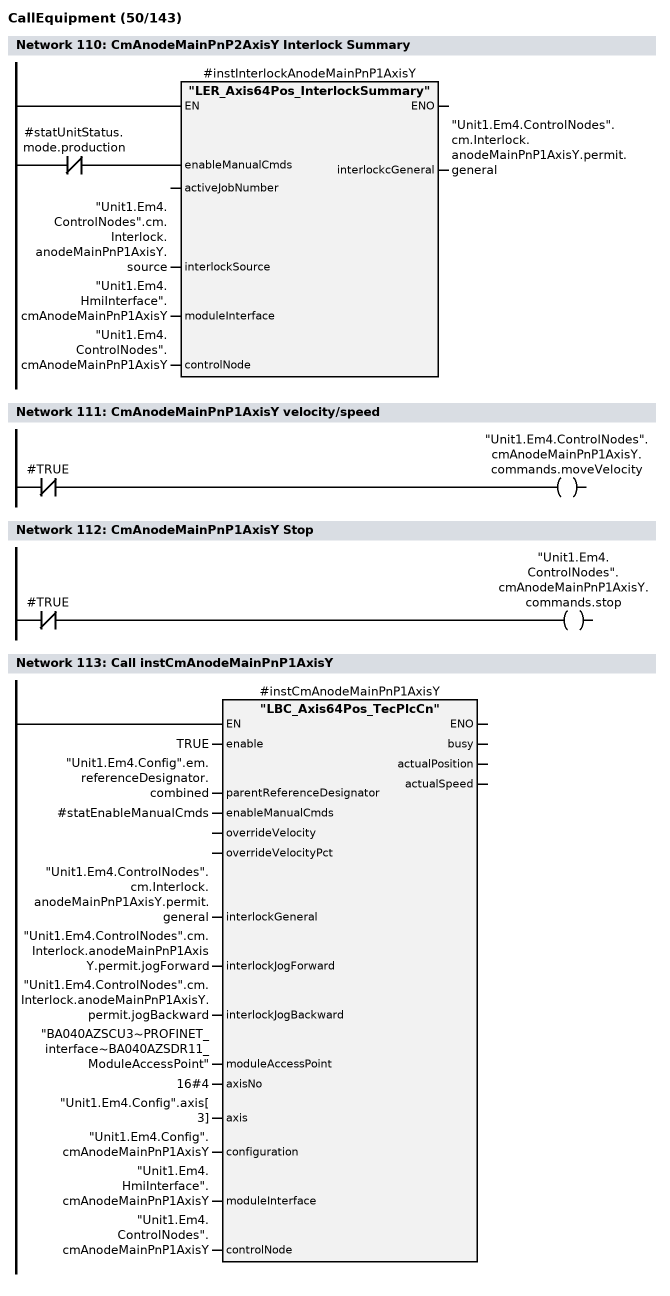
   RUNG wire#powerrail
      #instInterlockAnodeMainPnP1AxisY(enableManualCmds := wire#w1, activeJobNumber :=, interlockSource := "Unit1.Em4.ControlNodes".cm.Interlock.anodeMainPnP1AxisY.source, moduleInterface := "Unit1.Em4.HmiInterface".cmAnodeMainPnP1AxisY, controlNode := "Unit1.Em4.ControlNodes".cmAnodeMainPnP1AxisY, interlockcGeneral => "Unit1.Em4.ControlNodes".cm.Interlock.anodeMainPnP1AxisY.permit.general)
   END_RUNG
   RUNG wire#powerrail
      I_Contact( #statUnitStatus.mode.production )
   END_RUNG wire#w1
   // the same network as SCL:
   #instInterlockAnodeMainPnP1AxisY(enableManualCmds := NOT #statUnitStatus.mode.production,   // "LER_Axis64Pos_InterlockSummary"
                           interlockSource := "Unit1.Em4.ControlNodes".cm.Interlock.anodeMainPnP1AxisY.source,
                           moduleInterface := "Unit1.Em4.HmiInterface".cmAnodeMainPnP1AxisY,
                           controlNode := "Unit1.Em4.ControlNodes".cmAnodeMainPnP1AxisY,
                           interlockcGeneral => "Unit1.Em4.ControlNodes".cm.Interlock.anodeMainPnP1AxisY.permit.general);
END_REGION

REGION Network 111: CmAnodeMainPnP1AxisY velocity/speed
   RUNG wire#powerrail
      I_Contact( #TRUE )
      Coil( "Unit1.Em4.ControlNodes".cmAnodeMainPnP1AxisY.commands.moveVelocity )
   END_RUNG
   // the same network as SCL:
   "Unit1.Em4.ControlNodes".cmAnodeMainPnP1AxisY.commands.moveVelocity := NOT #TRUE;
END_REGION

REGION Network 112: CmAnodeMainPnP1AxisY Stop
   RUNG wire#powerrail
      I_Contact( #TRUE )
      Coil( "Unit1.Em4.ControlNodes".cmAnodeMainPnP1AxisY.commands.stop )
   END_RUNG
   // the same network as SCL:
   "Unit1.Em4.ControlNodes".cmAnodeMainPnP1AxisY.commands.stop := NOT #TRUE;
END_REGION

REGION Network 113: Call instCmAnodeMainPnP1AxisY
   RUNG wire#powerrail
      #instCmAnodeMainPnP1AxisY(enable := TRUE, parentReferenceDesignator := "Unit1.Em4.Config".em.referenceDesignator.combined, enableManualCmds := #statEnableManualCmds, overrideVelocity :=, overrideVelocityPct :=, interlockGeneral := "Unit1.Em4.ControlNodes".cm.Interlock.anodeMainPnP1AxisY.permit.general, interlockJogForward := "Unit1.Em4.ControlNodes".cm.Interlock.anodeMainPnP1AxisY.permit.jogForward, interlockJogBackward := "Unit1.Em4.ControlNodes".cm.Interlock.anodeMainPnP1AxisY.permit.jogBackward, moduleAccessPoint := "BA040AZSCU3~PROFINET_interface~BA040AZSDR11_ModuleAccessPoint", axisNo := 16#4, axis := "Unit1.Em4.Config".axis[3], configuration := "Unit1.Em4.Config".cmAnodeMainPnP1AxisY, moduleInterface := "Unit1.Em4.HmiInterface".cmAnodeMainPnP1AxisY, controlNode := "Unit1.Em4.ControlNodes".cmAnodeMainPnP1AxisY, busy =>, actualPosition =>, actualSpeed =>)
   END_RUNG
   // the same network as SCL:
   #instCmAnodeMainPnP1AxisY(enable := TRUE,   // "LBC_Axis64Pos_TecPlcCn"
                           parentReferenceDesignator := "Unit1.Em4.Config".em.referenceDesignator.combined,
                           enableManualCmds := #statEnableManualCmds,
                           interlockGeneral := "Unit1.Em4.ControlNodes".cm.Interlock.anodeMainPnP1AxisY.permit.general,
                           interlockJogForward := "Unit1.Em4.ControlNodes".cm.Interlock.anodeMainPnP1AxisY.permit.jogForward,
                           interlockJogBackward := "Unit1.Em4.ControlNodes".cm.Interlock.anodeMainPnP1AxisY.permit.jogBackward,
                           moduleAccessPoint := "BA040AZSCU3~PROFINET_interface~BA040AZSDR11_ModuleAccessPoint",
                           axisNo := 16#4,
                           axis := "Unit1.Em4.Config".axis[3],
                           configuration := "Unit1.Em4.Config".cmAnodeMainPnP1AxisY,
                           moduleInterface := "Unit1.Em4.HmiInterface".cmAnodeMainPnP1AxisY,
                           controlNode := "Unit1.Em4.ControlNodes".cmAnodeMainPnP1AxisY);
END_REGION

REGION Network 114: CmAnodeMainPnP1AxisY SoftCam
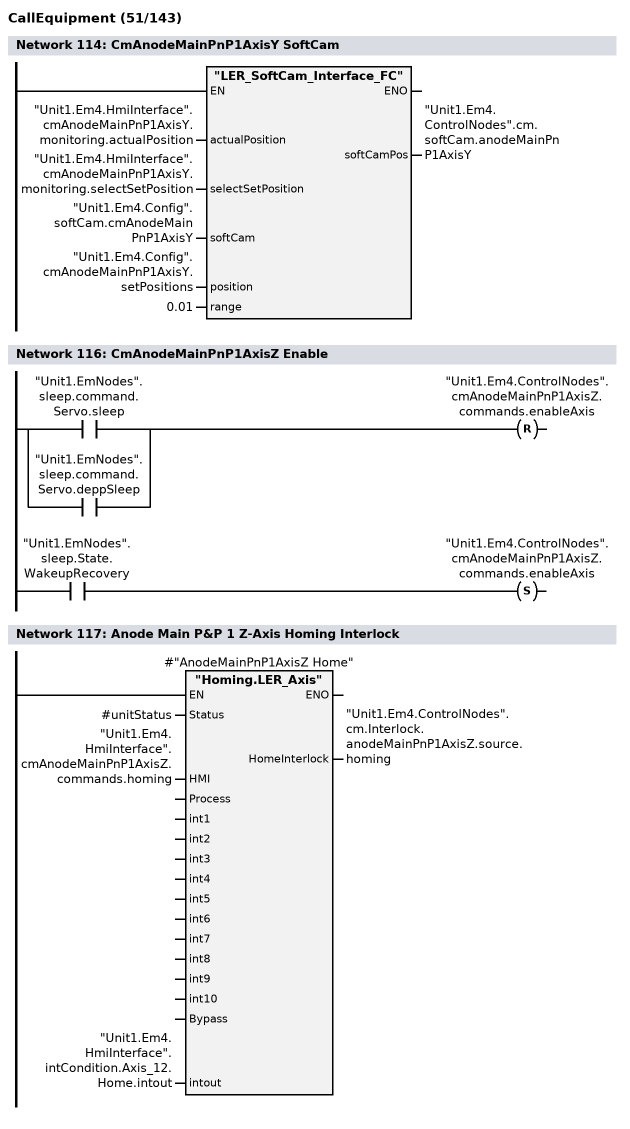
   RUNG wire#powerrail
      "LER_SoftCam_Interface_FC"(actualPosition := "Unit1.Em4.HmiInterface".cmAnodeMainPnP1AxisY.monitoring.actualPosition, selectSetPosition := "Unit1.Em4.HmiInterface".cmAnodeMainPnP1AxisY.monitoring.selectSetPosition, softCam := "Unit1.Em4.Config".softCam.cmAnodeMainPnP1AxisY, position := "Unit1.Em4.Config".cmAnodeMainPnP1AxisY.setPositions, range := 0.01, softCamPos => "Unit1.Em4.ControlNodes".cm.softCam.anodeMainPnP1AxisY)
   END_RUNG
   // the same network as SCL:
   "LER_SoftCam_Interface_FC"(actualPosition := "Unit1.Em4.HmiInterface".cmAnodeMainPnP1AxisY.monitoring.actualPosition,
                           selectSetPosition := "Unit1.Em4.HmiInterface".cmAnodeMainPnP1AxisY.monitoring.selectSetPosition,
                           softCam := "Unit1.Em4.Config".softCam.cmAnodeMainPnP1AxisY,
                           position := "Unit1.Em4.Config".cmAnodeMainPnP1AxisY.setPositions,
                           range := 0.01,
                           softCamPos => "Unit1.Em4.ControlNodes".cm.softCam.anodeMainPnP1AxisY);
END_REGION

REGION Network 116: CmAnodeMainPnP1AxisZ Enable
   RUNG wire#powerrail
      Contact( "Unit1.EmNodes".sleep.command.Servo.sleep )
      wire#w1
      R_Coil( "Unit1.Em4.ControlNodes".cmAnodeMainPnP1AxisZ.commands.enableAxis )
   END_RUNG
   RUNG wire#powerrail
      Contact( "Unit1.EmNodes".sleep.command.Servo.deppSleep )
   END_RUNG wire#w1
   RUNG wire#powerrail
      Contact( "Unit1.EmNodes".sleep.State.WakeupRecovery )
      S_Coil( "Unit1.Em4.ControlNodes".cmAnodeMainPnP1AxisZ.commands.enableAxis )
   END_RUNG
   // the same network as SCL:
   IF "Unit1.EmNodes".sleep.command.Servo.sleep OR "Unit1.EmNodes".sleep.command.Servo.deppSleep THEN
       "Unit1.Em4.ControlNodes".cmAnodeMainPnP1AxisZ.commands.enableAxis := FALSE;
   END_IF;
   IF "Unit1.EmNodes".sleep.State.WakeupRecovery THEN
       "Unit1.Em4.ControlNodes".cmAnodeMainPnP1AxisZ.commands.enableAxis := TRUE;
   END_IF;
END_REGION

REGION Network 117: Anode Main P&P 1 Z-Axis Homing Interlock
   RUNG wire#powerrail
      #"AnodeMainPnP1AxisZ Home"(Status := #unitStatus, HMI := "Unit1.Em4.HmiInterface".cmAnodeMainPnP1AxisZ.commands.homing, Process :=, int1 :=, int2 :=, int3 :=, int4 :=, int5 :=, int6 :=, int7 :=, int8 :=, int9 :=, int10 :=, Bypass :=, intout := "Unit1.Em4.HmiInterface".intCondition.Axis_12.Home.intout, HomeInterlock => "Unit1.Em4.ControlNodes".cm.Interlock.anodeMainPnP1AxisZ.source.homing)
   END_RUNG
   // the same network as SCL:
   #"AnodeMainPnP1AxisZ Home"(Status := #unitStatus,   // "Homing.LER_Axis"
                           HMI := "Unit1.Em4.HmiInterface".cmAnodeMainPnP1AxisZ.commands.homing,
                           intout := "Unit1.Em4.HmiInterface".intCondition.Axis_12.Home.intout,
                           HomeInterlock => "Unit1.Em4.ControlNodes".cm.Interlock.anodeMainPnP1AxisZ.source.homing);
END_REGION

REGION Network 118: CmAnodeMainPnP1AxisZ Position Absolute Jog
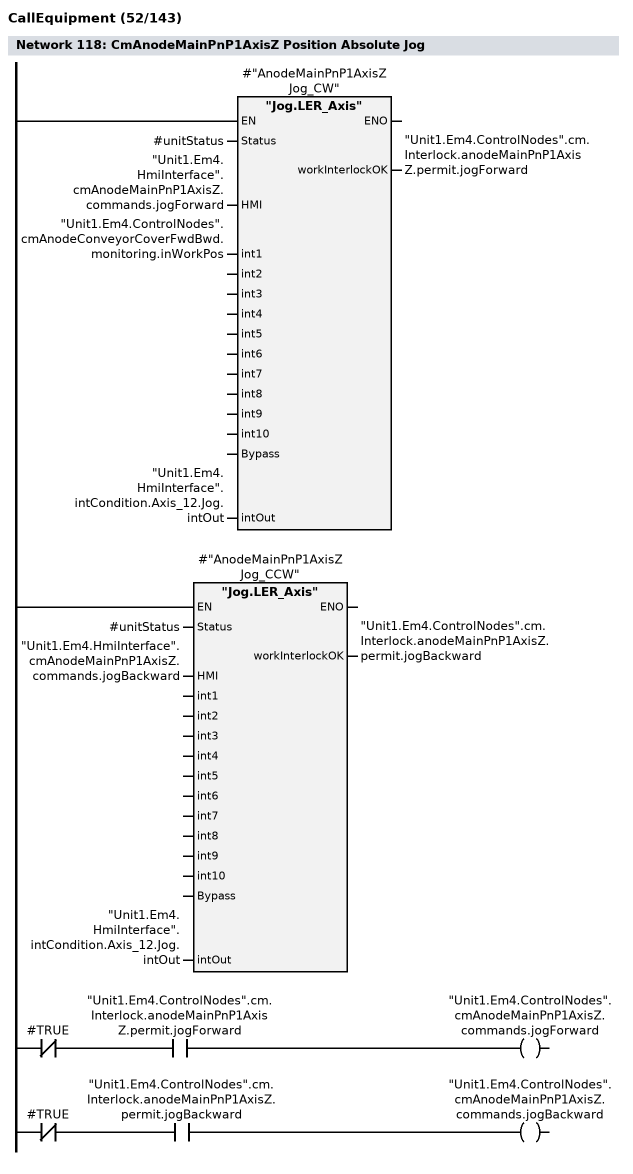
   RUNG wire#powerrail
      #"AnodeMainPnP1AxisZ Jog_CW"(Status := #unitStatus, HMI := "Unit1.Em4.HmiInterface".cmAnodeMainPnP1AxisZ.commands.jogForward, int1 := "Unit1.Em4.ControlNodes".cmAnodeConveyorCoverFwdBwd.monitoring.inWorkPos, int2 :=, int3 :=, int4 :=, int5 :=, int6 :=, int7 :=, int8 :=, int9 :=, int10 :=, Bypass :=, intOut := "Unit1.Em4.HmiInterface".intCondition.Axis_12.Jog.intOut, workInterlockOK => "Unit1.Em4.ControlNodes".cm.Interlock.anodeMainPnP1AxisZ.permit.jogForward)
   END_RUNG
   RUNG wire#powerrail
      #"AnodeMainPnP1AxisZ Jog_CCW"(Status := #unitStatus, HMI := "Unit1.Em4.HmiInterface".cmAnodeMainPnP1AxisZ.commands.jogBackward, int1 :=, int2 :=, int3 :=, int4 :=, int5 :=, int6 :=, int7 :=, int8 :=, int9 :=, int10 :=, Bypass :=, intOut := "Unit1.Em4.HmiInterface".intCondition.Axis_12.Jog.intOut, workInterlockOK => "Unit1.Em4.ControlNodes".cm.Interlock.anodeMainPnP1AxisZ.permit.jogBackward)
   END_RUNG
   RUNG wire#powerrail
      I_Contact( #TRUE )
      Contact( "Unit1.Em4.ControlNodes".cm.Interlock.anodeMainPnP1AxisZ.permit.jogForward )
      Coil( "Unit1.Em4.ControlNodes".cmAnodeMainPnP1AxisZ.commands.jogForward )
   END_RUNG
   RUNG wire#powerrail
      I_Contact( #TRUE )
      Contact( "Unit1.Em4.ControlNodes".cm.Interlock.anodeMainPnP1AxisZ.permit.jogBackward )
      Coil( "Unit1.Em4.ControlNodes".cmAnodeMainPnP1AxisZ.commands.jogBackward )
   END_RUNG
   // the same network as SCL:
   #"AnodeMainPnP1AxisZ Jog_CW"(Status := #unitStatus,   // "Jog.LER_Axis"
                           HMI := "Unit1.Em4.HmiInterface".cmAnodeMainPnP1AxisZ.commands.jogForward,
                           int1 := "Unit1.Em4.ControlNodes".cmAnodeConveyorCoverFwdBwd.monitoring.inWorkPos,
                           intOut := "Unit1.Em4.HmiInterface".intCondition.Axis_12.Jog.intOut,
                           workInterlockOK => "Unit1.Em4.ControlNodes".cm.Interlock.anodeMainPnP1AxisZ.permit.jogForward);
   #"AnodeMainPnP1AxisZ Jog_CCW"(Status := #unitStatus,   // "Jog.LER_Axis"
                           HMI := "Unit1.Em4.HmiInterface".cmAnodeMainPnP1AxisZ.commands.jogBackward,
                           intOut := "Unit1.Em4.HmiInterface".intCondition.Axis_12.Jog.intOut,
                           workInterlockOK => "Unit1.Em4.ControlNodes".cm.Interlock.anodeMainPnP1AxisZ.permit.jogBackward);
   "Unit1.Em4.ControlNodes".cmAnodeMainPnP1AxisZ.commands.jogForward := NOT #TRUE AND "Unit1.Em4.ControlNodes".cm.Interlock.anodeMainPnP1AxisZ.permit.jogForward;
   "Unit1.Em4.ControlNodes".cmAnodeMainPnP1AxisZ.commands.jogBackward := NOT #TRUE AND "Unit1.Em4.ControlNodes".cm.Interlock.anodeMainPnP1AxisZ.permit.jogBackward;
END_REGION

REGION Network 119: CmAnodeMainPnP1AxisZ Position Absolute Position0
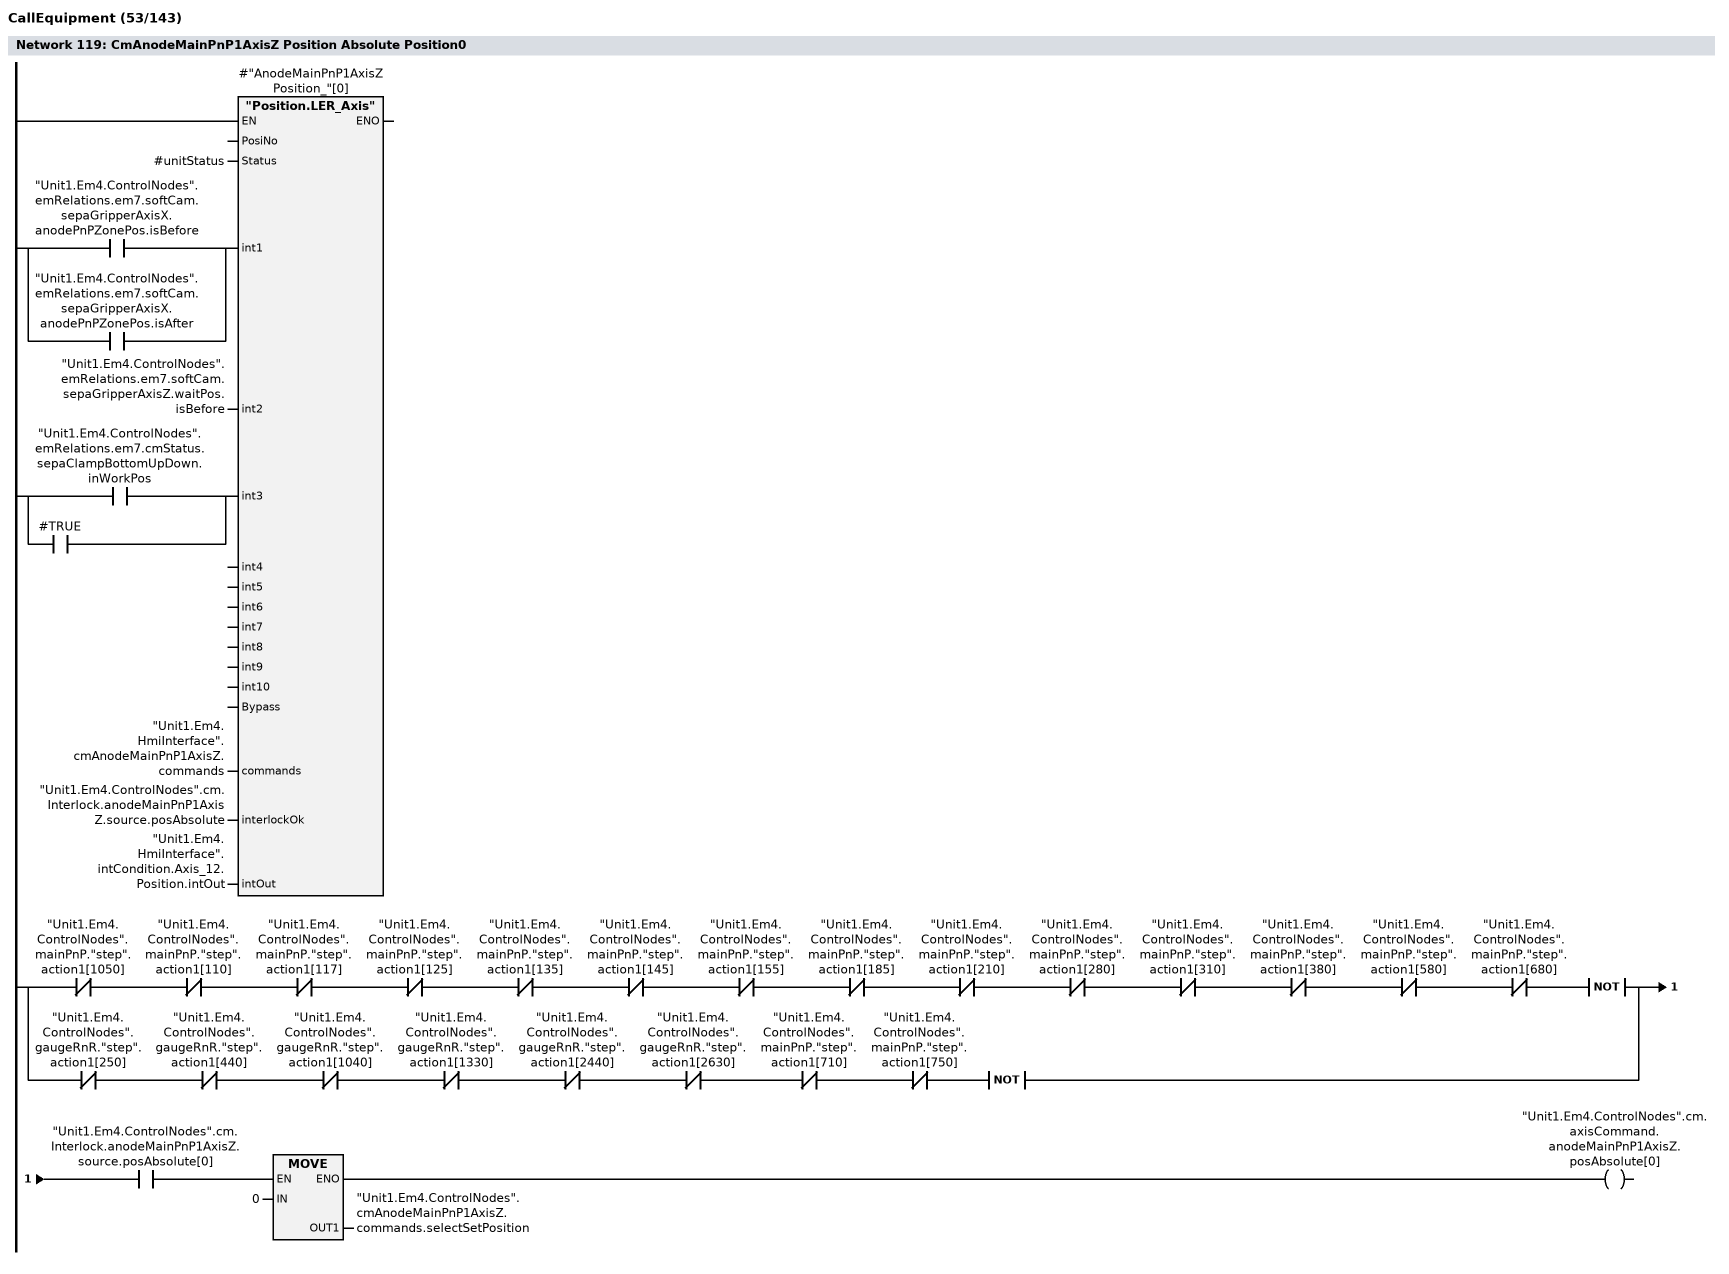
   RUNG wire#powerrail
      #"AnodeMainPnP1AxisZ Position_"[0](int1 := wire#w1, int3 := wire#w2, PosiNo :=, Status := #unitStatus, int2 := "Unit1.Em4.ControlNodes".emRelations.em7.softCam.sepaGripperAxisZ.waitPos.isBefore, int4 :=, int5 :=, int6 :=, int7 :=, int8 :=, int9 :=, int10 :=, Bypass :=, commands := "Unit1.Em4.HmiInterface".cmAnodeMainPnP1AxisZ.commands, interlockOk := "Unit1.Em4.ControlNodes".cm.Interlock.anodeMainPnP1AxisZ.source.posAbsolute, intOut := "Unit1.Em4.HmiInterface".intCondition.Axis_12.Position.intOut)
   END_RUNG
   RUNG wire#powerrail
      Contact( "Unit1.Em4.ControlNodes".emRelations.em7.softCam.sepaGripperAxisX.anodePnPZonePos.isBefore )
   END_RUNG wire#w1
   RUNG wire#powerrail
      Contact( "Unit1.Em4.ControlNodes".emRelations.em7.softCam.sepaGripperAxisX.anodePnPZonePos.isAfter )
   END_RUNG wire#w1
   RUNG wire#powerrail
      Contact( "Unit1.Em4.ControlNodes".emRelations.em7.cmStatus.sepaClampBottomUpDown.inWorkPos )
   END_RUNG wire#w2
   RUNG wire#powerrail
      Contact( #TRUE )
   END_RUNG wire#w2
   RUNG wire#powerrail
      I_Contact( "Unit1.Em4.ControlNodes".mainPnP."step".action1[1050] )
      I_Contact( "Unit1.Em4.ControlNodes".mainPnP."step".action1[110] )
      I_Contact( "Unit1.Em4.ControlNodes".mainPnP."step".action1[117] )
      I_Contact( "Unit1.Em4.ControlNodes".mainPnP."step".action1[125] )
      I_Contact( "Unit1.Em4.ControlNodes".mainPnP."step".action1[135] )
      I_Contact( "Unit1.Em4.ControlNodes".mainPnP."step".action1[145] )
      I_Contact( "Unit1.Em4.ControlNodes".mainPnP."step".action1[155] )
      I_Contact( "Unit1.Em4.ControlNodes".mainPnP."step".action1[185] )
      I_Contact( "Unit1.Em4.ControlNodes".mainPnP."step".action1[210] )
      I_Contact( "Unit1.Em4.ControlNodes".mainPnP."step".action1[280] )
      I_Contact( "Unit1.Em4.ControlNodes".mainPnP."step".action1[310] )
      I_Contact( "Unit1.Em4.ControlNodes".mainPnP."step".action1[380] )
      I_Contact( "Unit1.Em4.ControlNodes".mainPnP."step".action1[580] )
      I_Contact( "Unit1.Em4.ControlNodes".mainPnP."step".action1[680] )
      Not()
      wire#w3
      Contact( "Unit1.Em4.ControlNodes".cm.Interlock.anodeMainPnP1AxisZ.source.posAbsolute[0] )
      Move(in := 0, out1 => "Unit1.Em4.ControlNodes".cmAnodeMainPnP1AxisZ.commands.selectSetPosition)
      Coil( "Unit1.Em4.ControlNodes".cm.axisCommand.anodeMainPnP1AxisZ.posAbsolute[0] )
   END_RUNG
   RUNG wire#powerrail
      I_Contact( "Unit1.Em4.ControlNodes".gaugeRnR."step".action1[250] )
      I_Contact( "Unit1.Em4.ControlNodes".gaugeRnR."step".action1[440] )
      I_Contact( "Unit1.Em4.ControlNodes".gaugeRnR."step".action1[1040] )
      I_Contact( "Unit1.Em4.ControlNodes".gaugeRnR."step".action1[1330] )
      I_Contact( "Unit1.Em4.ControlNodes".gaugeRnR."step".action1[2440] )
      I_Contact( "Unit1.Em4.ControlNodes".gaugeRnR."step".action1[2630] )
      I_Contact( "Unit1.Em4.ControlNodes".mainPnP."step".action1[710] )
      I_Contact( "Unit1.Em4.ControlNodes".mainPnP."step".action1[750] )
      Not()
   END_RUNG wire#w3
   // the same network as SCL:
   #"AnodeMainPnP1AxisZ Position_"[0](Status := #unitStatus,   // "Position.LER_Axis"
                           int1 := "Unit1.Em4.ControlNodes".emRelations.em7.softCam.sepaGripperAxisX.anodePnPZonePos.isBefore OR "Unit1.Em4.ControlNodes".emRelations.em7.softCam.sepaGripperAxisX.anodePnPZonePos.isAfter,
                           int2 := "Unit1.Em4.ControlNodes".emRelations.em7.softCam.sepaGripperAxisZ.waitPos.isBefore,
                           int3 := "Unit1.Em4.ControlNodes".emRelations.em7.cmStatus.sepaClampBottomUpDown.inWorkPos OR #TRUE,
                           commands := "Unit1.Em4.HmiInterface".cmAnodeMainPnP1AxisZ.commands,
                           interlockOk := "Unit1.Em4.ControlNodes".cm.Interlock.anodeMainPnP1AxisZ.source.posAbsolute,
                           intOut := "Unit1.Em4.HmiInterface".intCondition.Axis_12.Position.intOut);
   #_w1 := (NOT (NOT "Unit1.Em4.ControlNodes".mainPnP."step".action1[1050] AND NOT "Unit1.Em4.ControlNodes".mainPnP."step".action1[110] AND NOT "Unit1.Em4.ControlNodes".mainPnP."step".action1[117] AND NOT "Unit1.Em4.ControlNodes".mainPnP."step".action1[125] AND NOT "Unit1.Em4.ControlNodes".mainPnP."step".action1[135] AND NOT "Unit1.Em4.ControlNodes".mainPnP."step".action1[145] AND NOT "Unit1.Em4.ControlNodes".mainPnP."step".action1[155] AND NOT "Unit1.Em4.ControlNodes".mainPnP."step".action1[185] AND NOT "Unit1.Em4.ControlNodes".mainPnP."step".action1[210] AND NOT "Unit1.Em4.ControlNodes".mainPnP."step".action1[280] AND NOT "Unit1.Em4.ControlNodes".mainPnP."step".action1[310] AND NOT "Unit1.Em4.ControlNodes".mainPnP."step".action1[380] AND NOT "Unit1.Em4.ControlNodes".mainPnP."step".action1[580] AND NOT "Unit1.Em4.ControlNodes".mainPnP."step".action1[680]) OR NOT (NOT "Unit1.Em4.ControlNodes".gaugeRnR."step".action1[250] AND NOT "Unit1.Em4.ControlNodes".gaugeRnR."step".action1[440] AND NOT "Unit1.Em4.ControlNodes".gaugeRnR."step".action1[1040] AND NOT "Unit1.Em4.ControlNodes".gaugeRnR."step".action1[1330] AND NOT "Unit1.Em4.ControlNodes".gaugeRnR."step".action1[2440] AND NOT "Unit1.Em4.ControlNodes".gaugeRnR."step".action1[2630] AND NOT "Unit1.Em4.ControlNodes".mainPnP."step".action1[710] AND NOT "Unit1.Em4.ControlNodes".mainPnP."step".action1[750])) AND "Unit1.Em4.ControlNodes".cm.Interlock.anodeMainPnP1AxisZ.source.posAbsolute[0];
   IF #_w1 THEN "Unit1.Em4.ControlNodes".cmAnodeMainPnP1AxisZ.commands.selectSetPosition := 0; END_IF;
   "Unit1.Em4.ControlNodes".cm.axisCommand.anodeMainPnP1AxisZ.posAbsolute[0] := #_w1;
END_REGION

REGION Network 120: CmAnodeMainPnP1AxisZ Position Absolute Position1
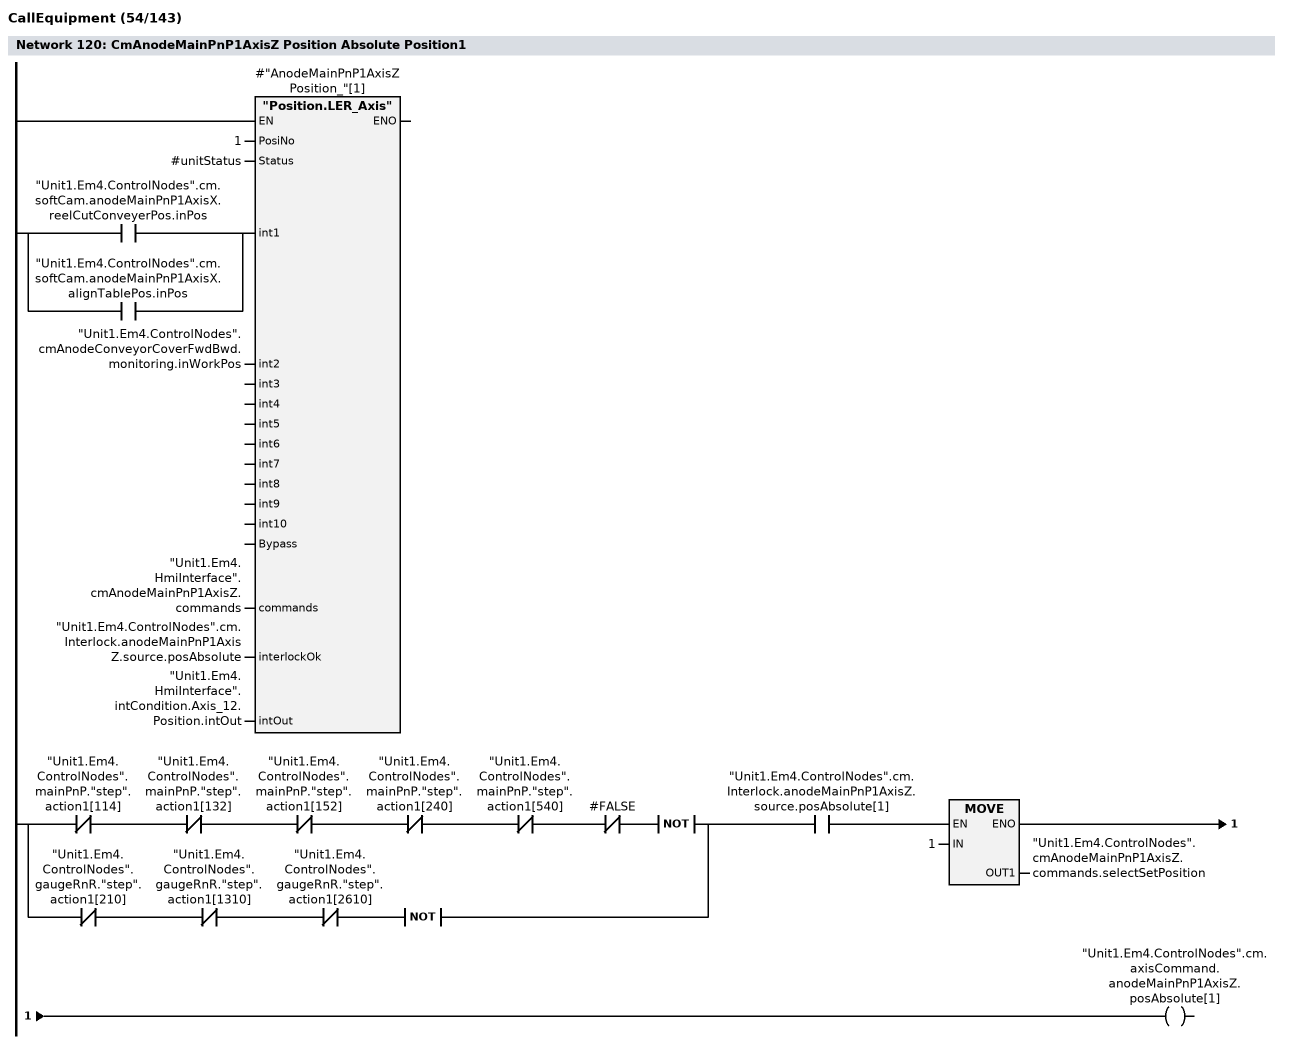
   RUNG wire#powerrail
      #"AnodeMainPnP1AxisZ Position_"[1](int1 := wire#w1, PosiNo := 1, Status := #unitStatus, int2 := "Unit1.Em4.ControlNodes".cmAnodeConveyorCoverFwdBwd.monitoring.inWorkPos, int3 :=, int4 :=, int5 :=, int6 :=, int7 :=, int8 :=, int9 :=, int10 :=, Bypass :=, commands := "Unit1.Em4.HmiInterface".cmAnodeMainPnP1AxisZ.commands, interlockOk := "Unit1.Em4.ControlNodes".cm.Interlock.anodeMainPnP1AxisZ.source.posAbsolute, intOut := "Unit1.Em4.HmiInterface".intCondition.Axis_12.Position.intOut)
   END_RUNG
   RUNG wire#powerrail
      Contact( "Unit1.Em4.ControlNodes".cm.softCam.anodeMainPnP1AxisX.reelCutConveyerPos.inPos )
   END_RUNG wire#w1
   RUNG wire#powerrail
      Contact( "Unit1.Em4.ControlNodes".cm.softCam.anodeMainPnP1AxisX.alignTablePos.inPos )
   END_RUNG wire#w1
   RUNG wire#powerrail
      I_Contact( "Unit1.Em4.ControlNodes".mainPnP."step".action1[114] )
      I_Contact( "Unit1.Em4.ControlNodes".mainPnP."step".action1[132] )
      I_Contact( "Unit1.Em4.ControlNodes".mainPnP."step".action1[152] )
      I_Contact( "Unit1.Em4.ControlNodes".mainPnP."step".action1[240] )
      I_Contact( "Unit1.Em4.ControlNodes".mainPnP."step".action1[540] )
      I_Contact( #FALSE )
      Not()
      wire#w2
      Contact( "Unit1.Em4.ControlNodes".cm.Interlock.anodeMainPnP1AxisZ.source.posAbsolute[1] )
      Move(in := 1, out1 => "Unit1.Em4.ControlNodes".cmAnodeMainPnP1AxisZ.commands.selectSetPosition)
      Coil( "Unit1.Em4.ControlNodes".cm.axisCommand.anodeMainPnP1AxisZ.posAbsolute[1] )
   END_RUNG
   RUNG wire#powerrail
      I_Contact( "Unit1.Em4.ControlNodes".gaugeRnR."step".action1[210] )
      I_Contact( "Unit1.Em4.ControlNodes".gaugeRnR."step".action1[1310] )
      I_Contact( "Unit1.Em4.ControlNodes".gaugeRnR."step".action1[2610] )
      Not()
   END_RUNG wire#w2
   // the same network as SCL:
   #"AnodeMainPnP1AxisZ Position_"[1](PosiNo := 1,   // "Position.LER_Axis"
                           Status := #unitStatus,
                           int1 := "Unit1.Em4.ControlNodes".cm.softCam.anodeMainPnP1AxisX.reelCutConveyerPos.inPos OR "Unit1.Em4.ControlNodes".cm.softCam.anodeMainPnP1AxisX.alignTablePos.inPos,
                           int2 := "Unit1.Em4.ControlNodes".cmAnodeConveyorCoverFwdBwd.monitoring.inWorkPos,
                           commands := "Unit1.Em4.HmiInterface".cmAnodeMainPnP1AxisZ.commands,
                           interlockOk := "Unit1.Em4.ControlNodes".cm.Interlock.anodeMainPnP1AxisZ.source.posAbsolute,
                           intOut := "Unit1.Em4.HmiInterface".intCondition.Axis_12.Position.intOut);
   #_w1 := (NOT (NOT "Unit1.Em4.ControlNodes".mainPnP."step".action1[114] AND NOT "Unit1.Em4.ControlNodes".mainPnP."step".action1[132] AND NOT "Unit1.Em4.ControlNodes".mainPnP."step".action1[152] AND NOT "Unit1.Em4.ControlNodes".mainPnP."step".action1[240] AND NOT "Unit1.Em4.ControlNodes".mainPnP."step".action1[540] AND NOT #FALSE) OR NOT (NOT "Unit1.Em4.ControlNodes".gaugeRnR."step".action1[210] AND NOT "Unit1.Em4.ControlNodes".gaugeRnR."step".action1[1310] AND NOT "Unit1.Em4.ControlNodes".gaugeRnR."step".action1[2610])) AND "Unit1.Em4.ControlNodes".cm.Interlock.anodeMainPnP1AxisZ.source.posAbsolute[1];
   IF #_w1 THEN "Unit1.Em4.ControlNodes".cmAnodeMainPnP1AxisZ.commands.selectSetPosition := 1; END_IF;
   "Unit1.Em4.ControlNodes".cm.axisCommand.anodeMainPnP1AxisZ.posAbsolute[1] := #_w1;
END_REGION

REGION Network 121: CmAnodeMainPnP1AxisZ Position Absolute Position2
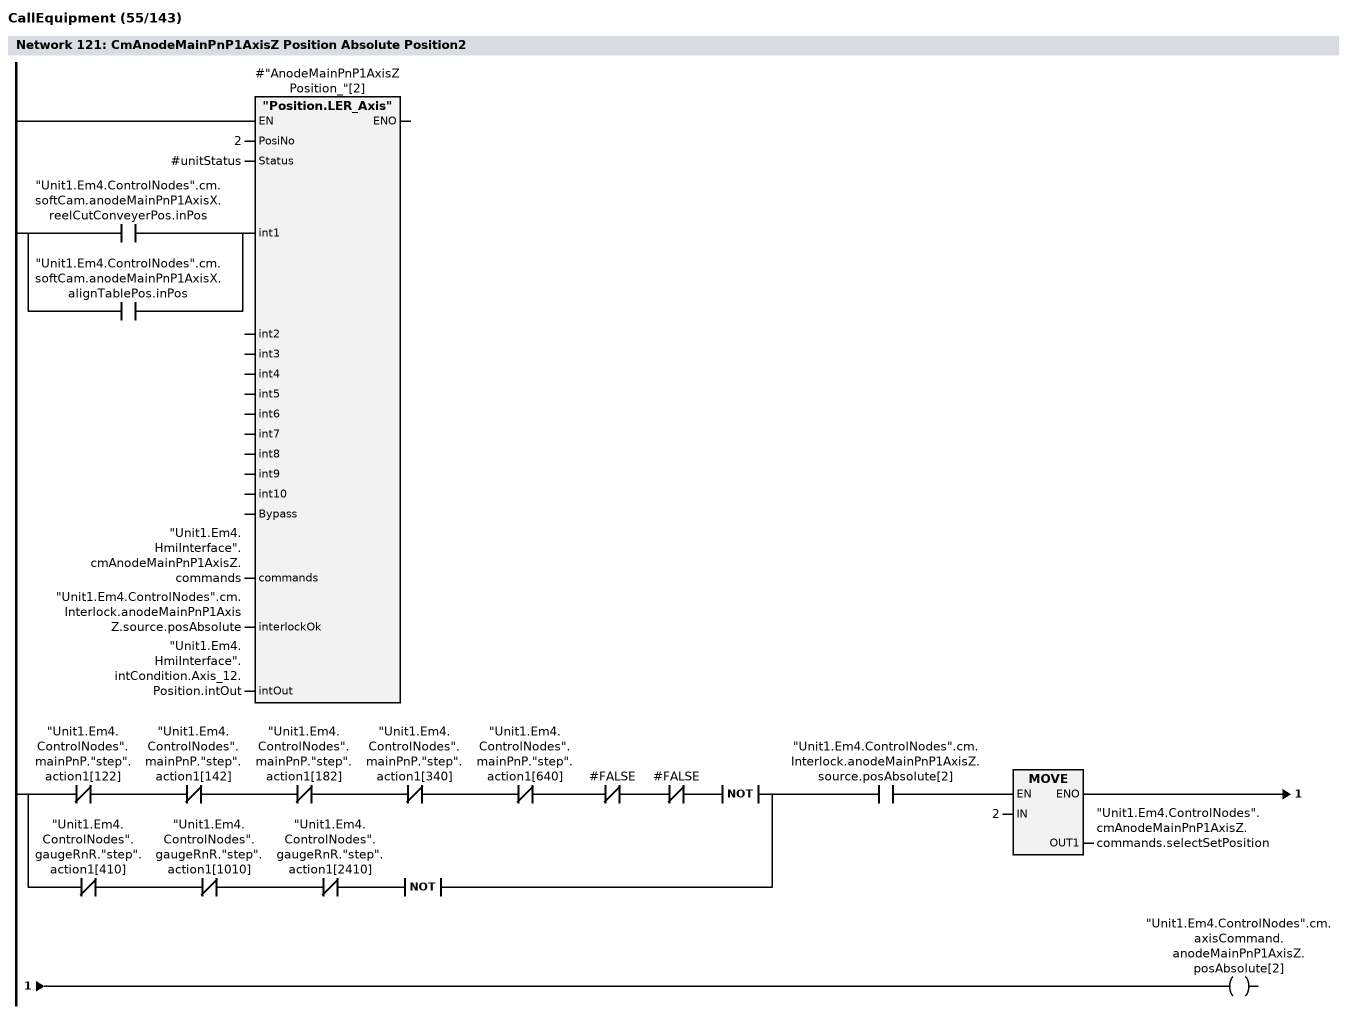
   RUNG wire#powerrail
      #"AnodeMainPnP1AxisZ Position_"[2](int1 := wire#w1, PosiNo := 2, Status := #unitStatus, int2 :=, int3 :=, int4 :=, int5 :=, int6 :=, int7 :=, int8 :=, int9 :=, int10 :=, Bypass :=, commands := "Unit1.Em4.HmiInterface".cmAnodeMainPnP1AxisZ.commands, interlockOk := "Unit1.Em4.ControlNodes".cm.Interlock.anodeMainPnP1AxisZ.source.posAbsolute, intOut := "Unit1.Em4.HmiInterface".intCondition.Axis_12.Position.intOut)
   END_RUNG
   RUNG wire#powerrail
      Contact( "Unit1.Em4.ControlNodes".cm.softCam.anodeMainPnP1AxisX.reelCutConveyerPos.inPos )
   END_RUNG wire#w1
   RUNG wire#powerrail
      Contact( "Unit1.Em4.ControlNodes".cm.softCam.anodeMainPnP1AxisX.alignTablePos.inPos )
   END_RUNG wire#w1
   RUNG wire#powerrail
      I_Contact( "Unit1.Em4.ControlNodes".mainPnP."step".action1[122] )
      I_Contact( "Unit1.Em4.ControlNodes".mainPnP."step".action1[142] )
      I_Contact( "Unit1.Em4.ControlNodes".mainPnP."step".action1[182] )
      I_Contact( "Unit1.Em4.ControlNodes".mainPnP."step".action1[340] )
      I_Contact( "Unit1.Em4.ControlNodes".mainPnP."step".action1[640] )
      I_Contact( #FALSE )
      I_Contact( #FALSE )
      Not()
      wire#w2
      Contact( "Unit1.Em4.ControlNodes".cm.Interlock.anodeMainPnP1AxisZ.source.posAbsolute[2] )
      Move(in := 2, out1 => "Unit1.Em4.ControlNodes".cmAnodeMainPnP1AxisZ.commands.selectSetPosition)
      Coil( "Unit1.Em4.ControlNodes".cm.axisCommand.anodeMainPnP1AxisZ.posAbsolute[2] )
   END_RUNG
   RUNG wire#powerrail
      I_Contact( "Unit1.Em4.ControlNodes".gaugeRnR."step".action1[410] )
      I_Contact( "Unit1.Em4.ControlNodes".gaugeRnR."step".action1[1010] )
      I_Contact( "Unit1.Em4.ControlNodes".gaugeRnR."step".action1[2410] )
      Not()
   END_RUNG wire#w2
   // the same network as SCL:
   #"AnodeMainPnP1AxisZ Position_"[2](PosiNo := 2,   // "Position.LER_Axis"
                           Status := #unitStatus,
                           int1 := "Unit1.Em4.ControlNodes".cm.softCam.anodeMainPnP1AxisX.reelCutConveyerPos.inPos OR "Unit1.Em4.ControlNodes".cm.softCam.anodeMainPnP1AxisX.alignTablePos.inPos,
                           commands := "Unit1.Em4.HmiInterface".cmAnodeMainPnP1AxisZ.commands,
                           interlockOk := "Unit1.Em4.ControlNodes".cm.Interlock.anodeMainPnP1AxisZ.source.posAbsolute,
                           intOut := "Unit1.Em4.HmiInterface".intCondition.Axis_12.Position.intOut);
   #_w1 := (NOT (NOT "Unit1.Em4.ControlNodes".mainPnP."step".action1[122] AND NOT "Unit1.Em4.ControlNodes".mainPnP."step".action1[142] AND NOT "Unit1.Em4.ControlNodes".mainPnP."step".action1[182] AND NOT "Unit1.Em4.ControlNodes".mainPnP."step".action1[340] AND NOT "Unit1.Em4.ControlNodes".mainPnP."step".action1[640] AND NOT #FALSE AND NOT #FALSE) OR NOT (NOT "Unit1.Em4.ControlNodes".gaugeRnR."step".action1[410] AND NOT "Unit1.Em4.ControlNodes".gaugeRnR."step".action1[1010] AND NOT "Unit1.Em4.ControlNodes".gaugeRnR."step".action1[2410])) AND "Unit1.Em4.ControlNodes".cm.Interlock.anodeMainPnP1AxisZ.source.posAbsolute[2];
   IF #_w1 THEN "Unit1.Em4.ControlNodes".cmAnodeMainPnP1AxisZ.commands.selectSetPosition := 2; END_IF;
   "Unit1.Em4.ControlNodes".cm.axisCommand.anodeMainPnP1AxisZ.posAbsolute[2] := #_w1;
END_REGION

REGION Network 122: CmAnodeMainPnP1AxisZ Position Absolute Position3
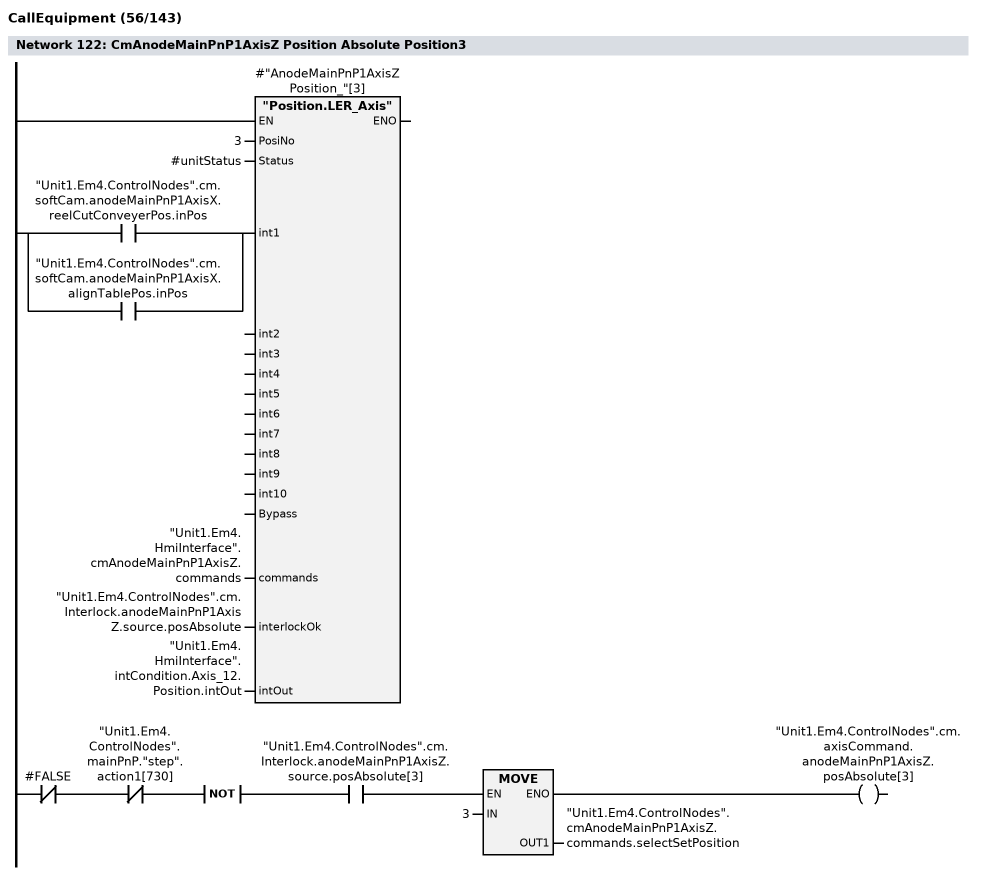
   RUNG wire#powerrail
      #"AnodeMainPnP1AxisZ Position_"[3](int1 := wire#w1, PosiNo := 3, Status := #unitStatus, int2 :=, int3 :=, int4 :=, int5 :=, int6 :=, int7 :=, int8 :=, int9 :=, int10 :=, Bypass :=, commands := "Unit1.Em4.HmiInterface".cmAnodeMainPnP1AxisZ.commands, interlockOk := "Unit1.Em4.ControlNodes".cm.Interlock.anodeMainPnP1AxisZ.source.posAbsolute, intOut := "Unit1.Em4.HmiInterface".intCondition.Axis_12.Position.intOut)
   END_RUNG
   RUNG wire#powerrail
      Contact( "Unit1.Em4.ControlNodes".cm.softCam.anodeMainPnP1AxisX.reelCutConveyerPos.inPos )
   END_RUNG wire#w1
   RUNG wire#powerrail
      Contact( "Unit1.Em4.ControlNodes".cm.softCam.anodeMainPnP1AxisX.alignTablePos.inPos )
   END_RUNG wire#w1
   RUNG wire#powerrail
      I_Contact( #FALSE )
      I_Contact( "Unit1.Em4.ControlNodes".mainPnP."step".action1[730] )
      Not()
      Contact( "Unit1.Em4.ControlNodes".cm.Interlock.anodeMainPnP1AxisZ.source.posAbsolute[3] )
      Move(in := 3, out1 => "Unit1.Em4.ControlNodes".cmAnodeMainPnP1AxisZ.commands.selectSetPosition)
      Coil( "Unit1.Em4.ControlNodes".cm.axisCommand.anodeMainPnP1AxisZ.posAbsolute[3] )
   END_RUNG
   // the same network as SCL:
   #"AnodeMainPnP1AxisZ Position_"[3](PosiNo := 3,   // "Position.LER_Axis"
                           Status := #unitStatus,
                           int1 := "Unit1.Em4.ControlNodes".cm.softCam.anodeMainPnP1AxisX.reelCutConveyerPos.inPos OR "Unit1.Em4.ControlNodes".cm.softCam.anodeMainPnP1AxisX.alignTablePos.inPos,
                           commands := "Unit1.Em4.HmiInterface".cmAnodeMainPnP1AxisZ.commands,
                           interlockOk := "Unit1.Em4.ControlNodes".cm.Interlock.anodeMainPnP1AxisZ.source.posAbsolute,
                           intOut := "Unit1.Em4.HmiInterface".intCondition.Axis_12.Position.intOut);
   #_w1 := NOT (NOT #FALSE AND NOT "Unit1.Em4.ControlNodes".mainPnP."step".action1[730]) AND "Unit1.Em4.ControlNodes".cm.Interlock.anodeMainPnP1AxisZ.source.posAbsolute[3];
   IF #_w1 THEN "Unit1.Em4.ControlNodes".cmAnodeMainPnP1AxisZ.commands.selectSetPosition := 3; END_IF;
   "Unit1.Em4.ControlNodes".cm.axisCommand.anodeMainPnP1AxisZ.posAbsolute[3] := #_w1;
END_REGION

REGION Network 123: CmAnodeMainPnP1AxisZ Position Absolute Position4
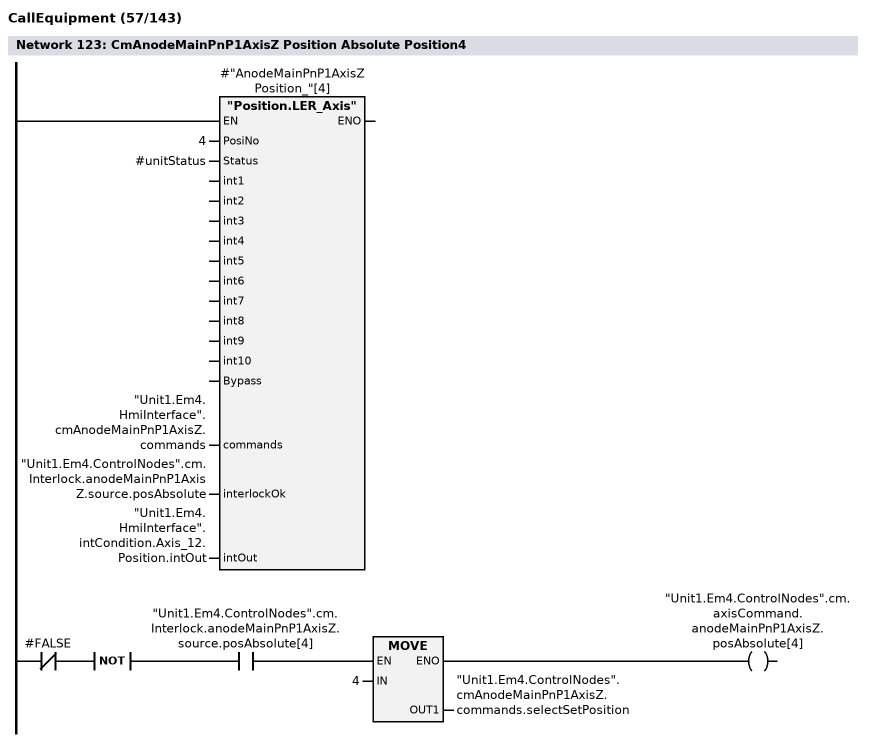
   RUNG wire#powerrail
      #"AnodeMainPnP1AxisZ Position_"[4](PosiNo := 4, Status := #unitStatus, int1 :=, int2 :=, int3 :=, int4 :=, int5 :=, int6 :=, int7 :=, int8 :=, int9 :=, int10 :=, Bypass :=, commands := "Unit1.Em4.HmiInterface".cmAnodeMainPnP1AxisZ.commands, interlockOk := "Unit1.Em4.ControlNodes".cm.Interlock.anodeMainPnP1AxisZ.source.posAbsolute, intOut := "Unit1.Em4.HmiInterface".intCondition.Axis_12.Position.intOut)
   END_RUNG
   RUNG wire#powerrail
      I_Contact( #FALSE )
      Not()
      Contact( "Unit1.Em4.ControlNodes".cm.Interlock.anodeMainPnP1AxisZ.source.posAbsolute[4] )
      Move(in := 4, out1 => "Unit1.Em4.ControlNodes".cmAnodeMainPnP1AxisZ.commands.selectSetPosition)
      Coil( "Unit1.Em4.ControlNodes".cm.axisCommand.anodeMainPnP1AxisZ.posAbsolute[4] )
   END_RUNG
   // the same network as SCL:
   #"AnodeMainPnP1AxisZ Position_"[4](PosiNo := 4,   // "Position.LER_Axis"
                           Status := #unitStatus,
                           commands := "Unit1.Em4.HmiInterface".cmAnodeMainPnP1AxisZ.commands,
                           interlockOk := "Unit1.Em4.ControlNodes".cm.Interlock.anodeMainPnP1AxisZ.source.posAbsolute,
                           intOut := "Unit1.Em4.HmiInterface".intCondition.Axis_12.Position.intOut);
   #_w1 := NOT (NOT #FALSE) AND "Unit1.Em4.ControlNodes".cm.Interlock.anodeMainPnP1AxisZ.source.posAbsolute[4];
   IF #_w1 THEN "Unit1.Em4.ControlNodes".cmAnodeMainPnP1AxisZ.commands.selectSetPosition := 4; END_IF;
   "Unit1.Em4.ControlNodes".cm.axisCommand.anodeMainPnP1AxisZ.posAbsolute[4] := #_w1;
END_REGION

REGION Network 124: CmAnodeMainPnP1AxisZ Position Absolute Position5
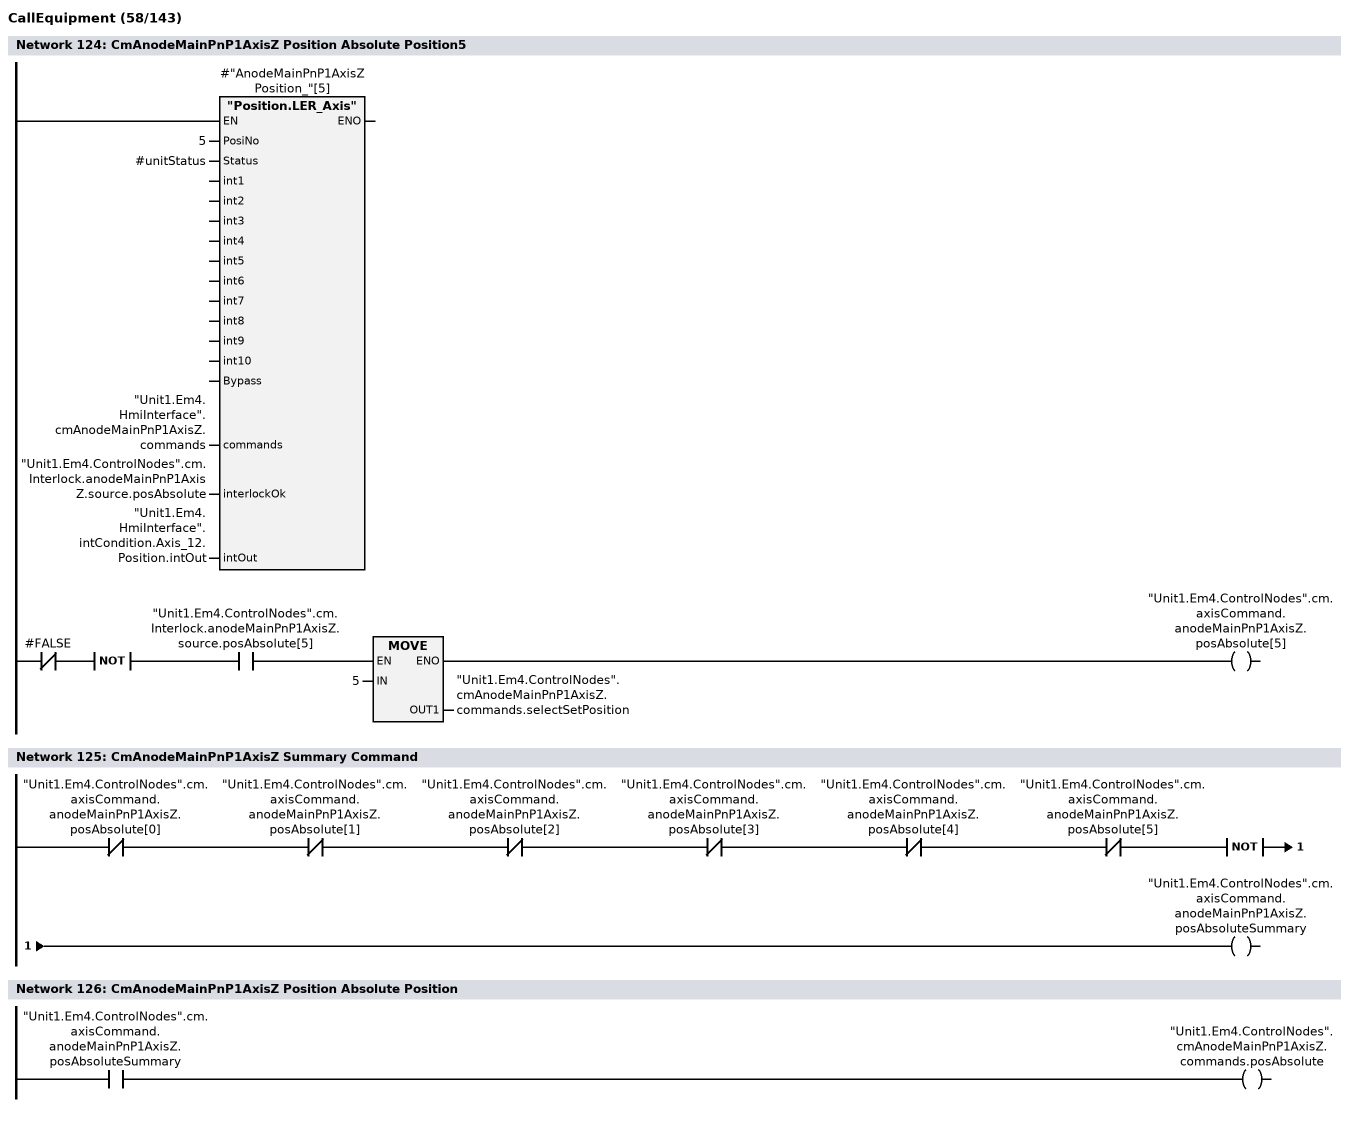
   RUNG wire#powerrail
      #"AnodeMainPnP1AxisZ Position_"[5](PosiNo := 5, Status := #unitStatus, int1 :=, int2 :=, int3 :=, int4 :=, int5 :=, int6 :=, int7 :=, int8 :=, int9 :=, int10 :=, Bypass :=, commands := "Unit1.Em4.HmiInterface".cmAnodeMainPnP1AxisZ.commands, interlockOk := "Unit1.Em4.ControlNodes".cm.Interlock.anodeMainPnP1AxisZ.source.posAbsolute, intOut := "Unit1.Em4.HmiInterface".intCondition.Axis_12.Position.intOut)
   END_RUNG
   RUNG wire#powerrail
      I_Contact( #FALSE )
      Not()
      Contact( "Unit1.Em4.ControlNodes".cm.Interlock.anodeMainPnP1AxisZ.source.posAbsolute[5] )
      Move(in := 5, out1 => "Unit1.Em4.ControlNodes".cmAnodeMainPnP1AxisZ.commands.selectSetPosition)
      Coil( "Unit1.Em4.ControlNodes".cm.axisCommand.anodeMainPnP1AxisZ.posAbsolute[5] )
   END_RUNG
   // the same network as SCL:
   #"AnodeMainPnP1AxisZ Position_"[5](PosiNo := 5,   // "Position.LER_Axis"
                           Status := #unitStatus,
                           commands := "Unit1.Em4.HmiInterface".cmAnodeMainPnP1AxisZ.commands,
                           interlockOk := "Unit1.Em4.ControlNodes".cm.Interlock.anodeMainPnP1AxisZ.source.posAbsolute,
                           intOut := "Unit1.Em4.HmiInterface".intCondition.Axis_12.Position.intOut);
   #_w1 := NOT (NOT #FALSE) AND "Unit1.Em4.ControlNodes".cm.Interlock.anodeMainPnP1AxisZ.source.posAbsolute[5];
   IF #_w1 THEN "Unit1.Em4.ControlNodes".cmAnodeMainPnP1AxisZ.commands.selectSetPosition := 5; END_IF;
   "Unit1.Em4.ControlNodes".cm.axisCommand.anodeMainPnP1AxisZ.posAbsolute[5] := #_w1;
END_REGION

REGION Network 125: CmAnodeMainPnP1AxisZ Summary Command
   RUNG wire#powerrail
      I_Contact( "Unit1.Em4.ControlNodes".cm.axisCommand.anodeMainPnP1AxisZ.posAbsolute[0] )
      I_Contact( "Unit1.Em4.ControlNodes".cm.axisCommand.anodeMainPnP1AxisZ.posAbsolute[1] )
      I_Contact( "Unit1.Em4.ControlNodes".cm.axisCommand.anodeMainPnP1AxisZ.posAbsolute[2] )
      I_Contact( "Unit1.Em4.ControlNodes".cm.axisCommand.anodeMainPnP1AxisZ.posAbsolute[3] )
      I_Contact( "Unit1.Em4.ControlNodes".cm.axisCommand.anodeMainPnP1AxisZ.posAbsolute[4] )
      I_Contact( "Unit1.Em4.ControlNodes".cm.axisCommand.anodeMainPnP1AxisZ.posAbsolute[5] )
      Not()
      Coil( "Unit1.Em4.ControlNodes".cm.axisCommand.anodeMainPnP1AxisZ.posAbsoluteSummary )
   END_RUNG
   // the same network as SCL:
   "Unit1.Em4.ControlNodes".cm.axisCommand.anodeMainPnP1AxisZ.posAbsoluteSummary := NOT (NOT "Unit1.Em4.ControlNodes".cm.axisCommand.anodeMainPnP1AxisZ.posAbsolute[0] AND NOT "Unit1.Em4.ControlNodes".cm.axisCommand.anodeMainPnP1AxisZ.posAbsolute[1] AND NOT "Unit1.Em4.ControlNodes".cm.axisCommand.anodeMainPnP1AxisZ.posAbsolute[2] AND NOT "Unit1.Em4.ControlNodes".cm.axisCommand.anodeMainPnP1AxisZ.posAbsolute[3] AND NOT "Unit1.Em4.ControlNodes".cm.axisCommand.anodeMainPnP1AxisZ.posAbsolute[4] AND NOT "Unit1.Em4.ControlNodes".cm.axisCommand.anodeMainPnP1AxisZ.posAbsolute[5]);
END_REGION

REGION Network 126: CmAnodeMainPnP1AxisZ Position Absolute Position
   RUNG wire#powerrail
      Contact( "Unit1.Em4.ControlNodes".cm.axisCommand.anodeMainPnP1AxisZ.posAbsoluteSummary )
      Coil( "Unit1.Em4.ControlNodes".cmAnodeMainPnP1AxisZ.commands.posAbsolute )
   END_RUNG
   // the same network as SCL:
   "Unit1.Em4.ControlNodes".cmAnodeMainPnP1AxisZ.commands.posAbsolute := "Unit1.Em4.ControlNodes".cm.axisCommand.anodeMainPnP1AxisZ.posAbsoluteSummary;
END_REGION

REGION Network 127: CmAnodeMainPnP1AxisZ Interlock Summary
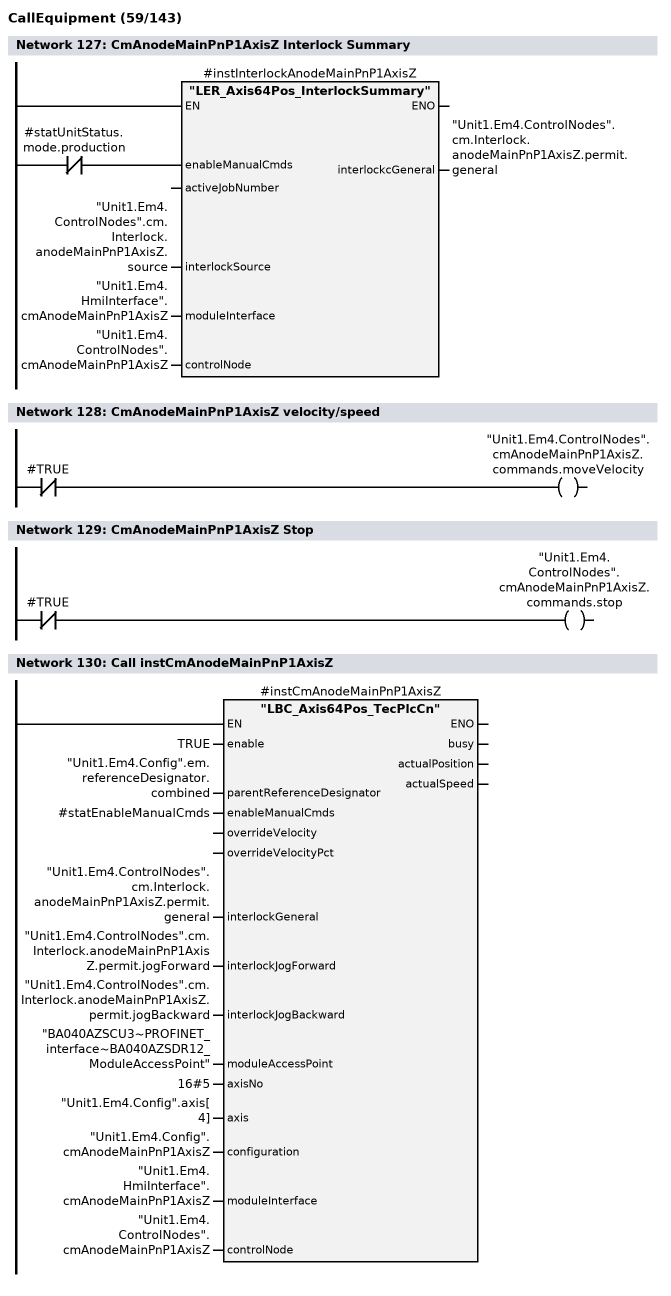
   RUNG wire#powerrail
      #instInterlockAnodeMainPnP1AxisZ(enableManualCmds := wire#w1, activeJobNumber :=, interlockSource := "Unit1.Em4.ControlNodes".cm.Interlock.anodeMainPnP1AxisZ.source, moduleInterface := "Unit1.Em4.HmiInterface".cmAnodeMainPnP1AxisZ, controlNode := "Unit1.Em4.ControlNodes".cmAnodeMainPnP1AxisZ, interlockcGeneral => "Unit1.Em4.ControlNodes".cm.Interlock.anodeMainPnP1AxisZ.permit.general)
   END_RUNG
   RUNG wire#powerrail
      I_Contact( #statUnitStatus.mode.production )
   END_RUNG wire#w1
   // the same network as SCL:
   #instInterlockAnodeMainPnP1AxisZ(enableManualCmds := NOT #statUnitStatus.mode.production,   // "LER_Axis64Pos_InterlockSummary"
                           interlockSource := "Unit1.Em4.ControlNodes".cm.Interlock.anodeMainPnP1AxisZ.source,
                           moduleInterface := "Unit1.Em4.HmiInterface".cmAnodeMainPnP1AxisZ,
                           controlNode := "Unit1.Em4.ControlNodes".cmAnodeMainPnP1AxisZ,
                           interlockcGeneral => "Unit1.Em4.ControlNodes".cm.Interlock.anodeMainPnP1AxisZ.permit.general);
END_REGION

REGION Network 128: CmAnodeMainPnP1AxisZ velocity/speed
   RUNG wire#powerrail
      I_Contact( #TRUE )
      Coil( "Unit1.Em4.ControlNodes".cmAnodeMainPnP1AxisZ.commands.moveVelocity )
   END_RUNG
   // the same network as SCL:
   "Unit1.Em4.ControlNodes".cmAnodeMainPnP1AxisZ.commands.moveVelocity := NOT #TRUE;
END_REGION

REGION Network 129: CmAnodeMainPnP1AxisZ Stop
   RUNG wire#powerrail
      I_Contact( #TRUE )
      Coil( "Unit1.Em4.ControlNodes".cmAnodeMainPnP1AxisZ.commands.stop )
   END_RUNG
   // the same network as SCL:
   "Unit1.Em4.ControlNodes".cmAnodeMainPnP1AxisZ.commands.stop := NOT #TRUE;
END_REGION

REGION Network 130: Call instCmAnodeMainPnP1AxisZ
   RUNG wire#powerrail
      #instCmAnodeMainPnP1AxisZ(enable := TRUE, parentReferenceDesignator := "Unit1.Em4.Config".em.referenceDesignator.combined, enableManualCmds := #statEnableManualCmds, overrideVelocity :=, overrideVelocityPct :=, interlockGeneral := "Unit1.Em4.ControlNodes".cm.Interlock.anodeMainPnP1AxisZ.permit.general, interlockJogForward := "Unit1.Em4.ControlNodes".cm.Interlock.anodeMainPnP1AxisZ.permit.jogForward, interlockJogBackward := "Unit1.Em4.ControlNodes".cm.Interlock.anodeMainPnP1AxisZ.permit.jogBackward, moduleAccessPoint := "BA040AZSCU3~PROFINET_interface~BA040AZSDR12_ModuleAccessPoint", axisNo := 16#5, axis := "Unit1.Em4.Config".axis[4], configuration := "Unit1.Em4.Config".cmAnodeMainPnP1AxisZ, moduleInterface := "Unit1.Em4.HmiInterface".cmAnodeMainPnP1AxisZ, controlNode := "Unit1.Em4.ControlNodes".cmAnodeMainPnP1AxisZ, busy =>, actualPosition =>, actualSpeed =>)
   END_RUNG
   // the same network as SCL:
   #instCmAnodeMainPnP1AxisZ(enable := TRUE,   // "LBC_Axis64Pos_TecPlcCn"
                           parentReferenceDesignator := "Unit1.Em4.Config".em.referenceDesignator.combined,
                           enableManualCmds := #statEnableManualCmds,
                           interlockGeneral := "Unit1.Em4.ControlNodes".cm.Interlock.anodeMainPnP1AxisZ.permit.general,
                           interlockJogForward := "Unit1.Em4.ControlNodes".cm.Interlock.anodeMainPnP1AxisZ.permit.jogForward,
                           interlockJogBackward := "Unit1.Em4.ControlNodes".cm.Interlock.anodeMainPnP1AxisZ.permit.jogBackward,
                           moduleAccessPoint := "BA040AZSCU3~PROFINET_interface~BA040AZSDR12_ModuleAccessPoint",
                           axisNo := 16#5,
                           axis := "Unit1.Em4.Config".axis[4],
                           configuration := "Unit1.Em4.Config".cmAnodeMainPnP1AxisZ,
                           moduleInterface := "Unit1.Em4.HmiInterface".cmAnodeMainPnP1AxisZ,
                           controlNode := "Unit1.Em4.ControlNodes".cmAnodeMainPnP1AxisZ);
END_REGION

REGION Network 131: CmAnodeMainPnP1AxisY SoftCam
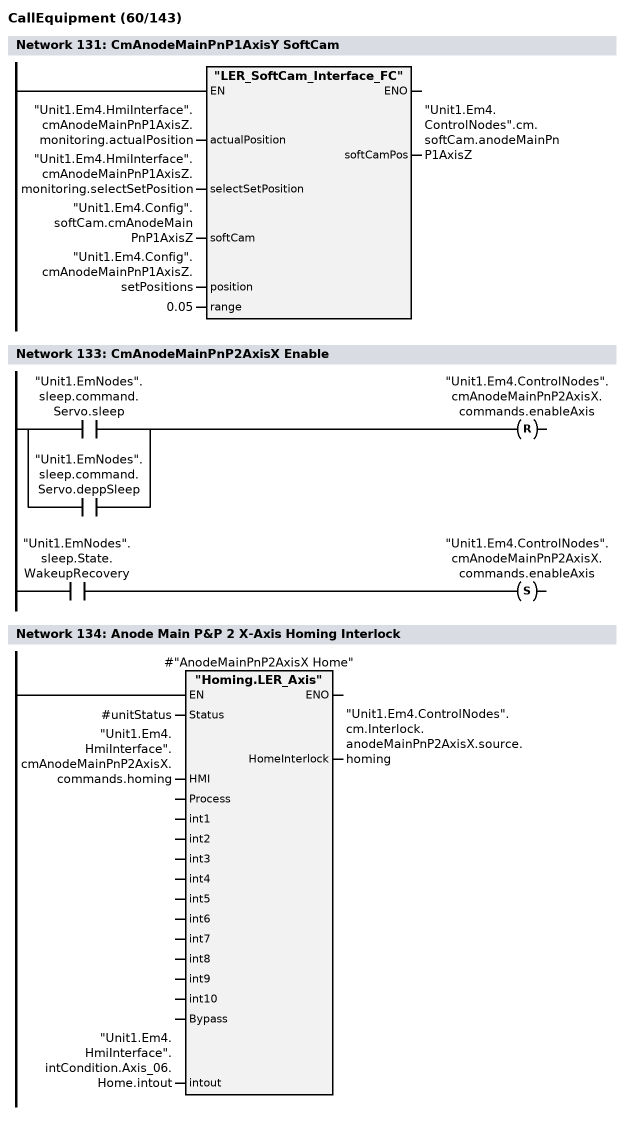
   RUNG wire#powerrail
      "LER_SoftCam_Interface_FC"(actualPosition := "Unit1.Em4.HmiInterface".cmAnodeMainPnP1AxisZ.monitoring.actualPosition, selectSetPosition := "Unit1.Em4.HmiInterface".cmAnodeMainPnP1AxisZ.monitoring.selectSetPosition, softCam := "Unit1.Em4.Config".softCam.cmAnodeMainPnP1AxisZ, position := "Unit1.Em4.Config".cmAnodeMainPnP1AxisZ.setPositions, range := 0.05, softCamPos => "Unit1.Em4.ControlNodes".cm.softCam.anodeMainPnP1AxisZ)
   END_RUNG
   // the same network as SCL:
   "LER_SoftCam_Interface_FC"(actualPosition := "Unit1.Em4.HmiInterface".cmAnodeMainPnP1AxisZ.monitoring.actualPosition,
                           selectSetPosition := "Unit1.Em4.HmiInterface".cmAnodeMainPnP1AxisZ.monitoring.selectSetPosition,
                           softCam := "Unit1.Em4.Config".softCam.cmAnodeMainPnP1AxisZ,
                           position := "Unit1.Em4.Config".cmAnodeMainPnP1AxisZ.setPositions,
                           range := 0.05,
                           softCamPos => "Unit1.Em4.ControlNodes".cm.softCam.anodeMainPnP1AxisZ);
END_REGION

REGION Network 133: CmAnodeMainPnP2AxisX Enable
   RUNG wire#powerrail
      Contact( "Unit1.EmNodes".sleep.command.Servo.sleep )
      wire#w1
      R_Coil( "Unit1.Em4.ControlNodes".cmAnodeMainPnP2AxisX.commands.enableAxis )
   END_RUNG
   RUNG wire#powerrail
      Contact( "Unit1.EmNodes".sleep.command.Servo.deppSleep )
   END_RUNG wire#w1
   RUNG wire#powerrail
      Contact( "Unit1.EmNodes".sleep.State.WakeupRecovery )
      S_Coil( "Unit1.Em4.ControlNodes".cmAnodeMainPnP2AxisX.commands.enableAxis )
   END_RUNG
   // the same network as SCL:
   IF "Unit1.EmNodes".sleep.command.Servo.sleep OR "Unit1.EmNodes".sleep.command.Servo.deppSleep THEN
       "Unit1.Em4.ControlNodes".cmAnodeMainPnP2AxisX.commands.enableAxis := FALSE;
   END_IF;
   IF "Unit1.EmNodes".sleep.State.WakeupRecovery THEN
       "Unit1.Em4.ControlNodes".cmAnodeMainPnP2AxisX.commands.enableAxis := TRUE;
   END_IF;
END_REGION

REGION Network 134: Anode Main P&P 2 X-Axis Homing Interlock
   RUNG wire#powerrail
      #"AnodeMainPnP2AxisX Home"(Status := #unitStatus, HMI := "Unit1.Em4.HmiInterface".cmAnodeMainPnP2AxisX.commands.homing, Process :=, int1 :=, int2 :=, int3 :=, int4 :=, int5 :=, int6 :=, int7 :=, int8 :=, int9 :=, int10 :=, Bypass :=, intout := "Unit1.Em4.HmiInterface".intCondition.Axis_06.Home.intout, HomeInterlock => "Unit1.Em4.ControlNodes".cm.Interlock.anodeMainPnP2AxisX.source.homing)
   END_RUNG
   // the same network as SCL:
   #"AnodeMainPnP2AxisX Home"(Status := #unitStatus,   // "Homing.LER_Axis"
                           HMI := "Unit1.Em4.HmiInterface".cmAnodeMainPnP2AxisX.commands.homing,
                           intout := "Unit1.Em4.HmiInterface".intCondition.Axis_06.Home.intout,
                           HomeInterlock => "Unit1.Em4.ControlNodes".cm.Interlock.anodeMainPnP2AxisX.source.homing);
END_REGION

REGION Network 135: CmAnodeMainPnP2AxisX Position Absolute Jog
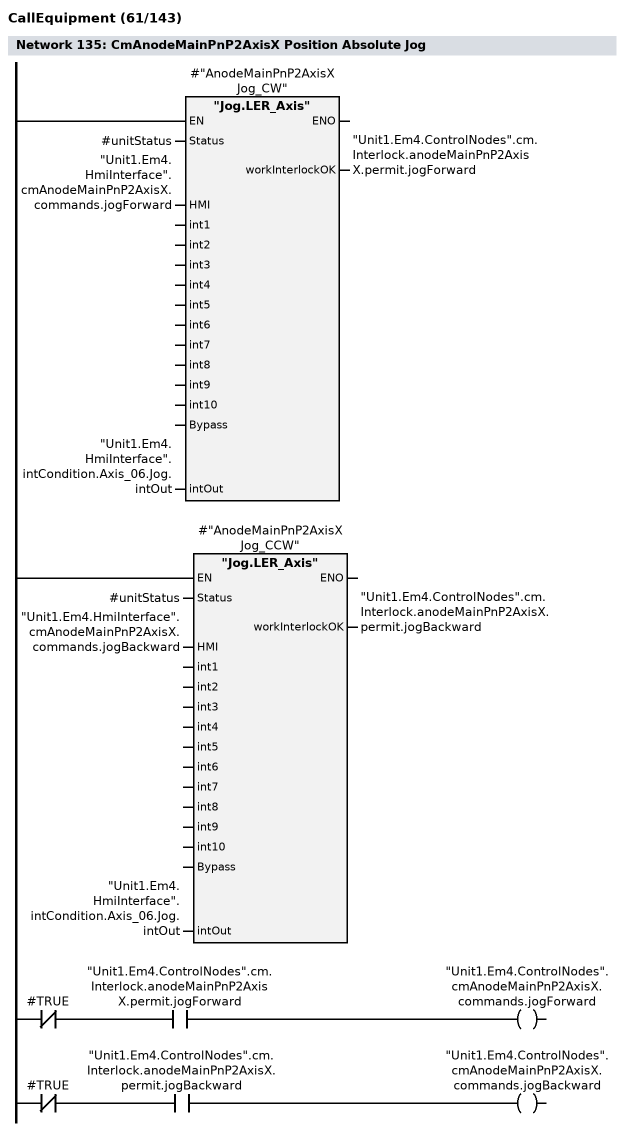
   RUNG wire#powerrail
      #"AnodeMainPnP2AxisX Jog_CW"(Status := #unitStatus, HMI := "Unit1.Em4.HmiInterface".cmAnodeMainPnP2AxisX.commands.jogForward, int1 :=, int2 :=, int3 :=, int4 :=, int5 :=, int6 :=, int7 :=, int8 :=, int9 :=, int10 :=, Bypass :=, intOut := "Unit1.Em4.HmiInterface".intCondition.Axis_06.Jog.intOut, workInterlockOK => "Unit1.Em4.ControlNodes".cm.Interlock.anodeMainPnP2AxisX.permit.jogForward)
   END_RUNG
   RUNG wire#powerrail
      #"AnodeMainPnP2AxisX Jog_CCW"(Status := #unitStatus, HMI := "Unit1.Em4.HmiInterface".cmAnodeMainPnP2AxisX.commands.jogBackward, int1 :=, int2 :=, int3 :=, int4 :=, int5 :=, int6 :=, int7 :=, int8 :=, int9 :=, int10 :=, Bypass :=, intOut := "Unit1.Em4.HmiInterface".intCondition.Axis_06.Jog.intOut, workInterlockOK => "Unit1.Em4.ControlNodes".cm.Interlock.anodeMainPnP2AxisX.permit.jogBackward)
   END_RUNG
   RUNG wire#powerrail
      I_Contact( #TRUE )
      Contact( "Unit1.Em4.ControlNodes".cm.Interlock.anodeMainPnP2AxisX.permit.jogForward )
      Coil( "Unit1.Em4.ControlNodes".cmAnodeMainPnP2AxisX.commands.jogForward )
   END_RUNG
   RUNG wire#powerrail
      I_Contact( #TRUE )
      Contact( "Unit1.Em4.ControlNodes".cm.Interlock.anodeMainPnP2AxisX.permit.jogBackward )
      Coil( "Unit1.Em4.ControlNodes".cmAnodeMainPnP2AxisX.commands.jogBackward )
   END_RUNG
   // the same network as SCL:
   #"AnodeMainPnP2AxisX Jog_CW"(Status := #unitStatus,   // "Jog.LER_Axis"
                           HMI := "Unit1.Em4.HmiInterface".cmAnodeMainPnP2AxisX.commands.jogForward,
                           intOut := "Unit1.Em4.HmiInterface".intCondition.Axis_06.Jog.intOut,
                           workInterlockOK => "Unit1.Em4.ControlNodes".cm.Interlock.anodeMainPnP2AxisX.permit.jogForward);
   #"AnodeMainPnP2AxisX Jog_CCW"(Status := #unitStatus,   // "Jog.LER_Axis"
                           HMI := "Unit1.Em4.HmiInterface".cmAnodeMainPnP2AxisX.commands.jogBackward,
                           intOut := "Unit1.Em4.HmiInterface".intCondition.Axis_06.Jog.intOut,
                           workInterlockOK => "Unit1.Em4.ControlNodes".cm.Interlock.anodeMainPnP2AxisX.permit.jogBackward);
   "Unit1.Em4.ControlNodes".cmAnodeMainPnP2AxisX.commands.jogForward := NOT #TRUE AND "Unit1.Em4.ControlNodes".cm.Interlock.anodeMainPnP2AxisX.permit.jogForward;
   "Unit1.Em4.ControlNodes".cmAnodeMainPnP2AxisX.commands.jogBackward := NOT #TRUE AND "Unit1.Em4.ControlNodes".cm.Interlock.anodeMainPnP2AxisX.permit.jogBackward;
END_REGION

REGION Network 136: CmAnodeMainPnP2AxisX Position Absolute Position0
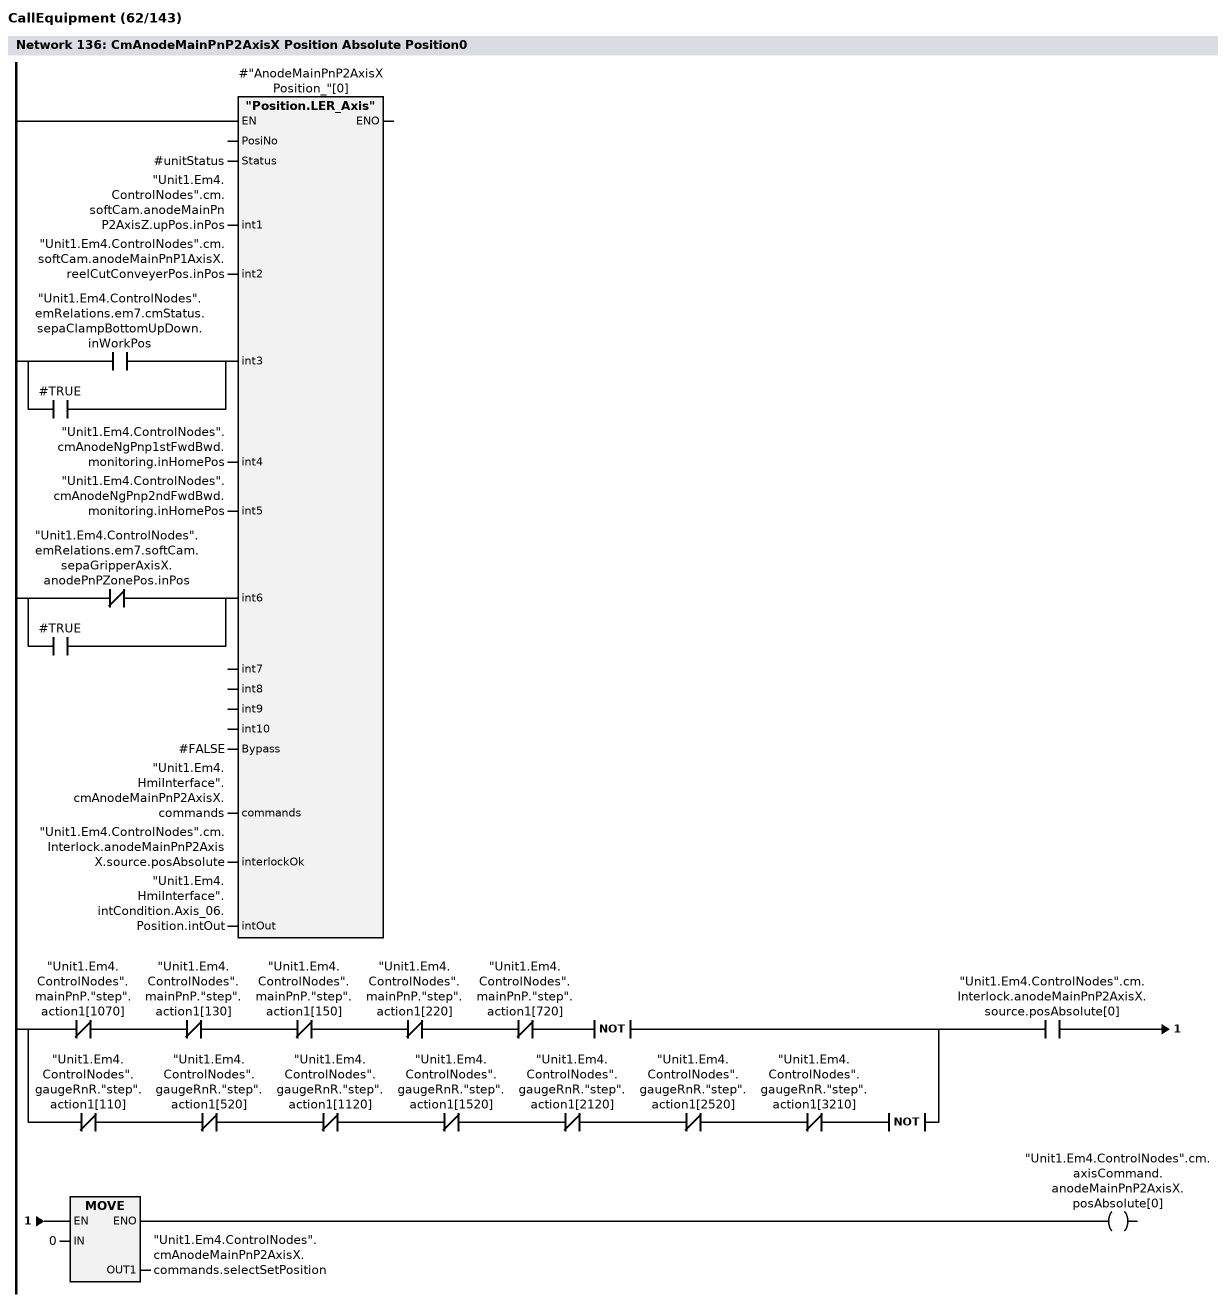
   RUNG wire#powerrail
      #"AnodeMainPnP2AxisX Position_"[0](int3 := wire#w1, int6 := wire#w2, PosiNo :=, Status := #unitStatus, int1 := "Unit1.Em4.ControlNodes".cm.softCam.anodeMainPnP2AxisZ.upPos.inPos, int2 := "Unit1.Em4.ControlNodes".cm.softCam.anodeMainPnP1AxisX.reelCutConveyerPos.inPos, int4 := "Unit1.Em4.ControlNodes".cmAnodeNgPnp1stFwdBwd.monitoring.inHomePos, int5 := "Unit1.Em4.ControlNodes".cmAnodeNgPnp2ndFwdBwd.monitoring.inHomePos, int7 :=, int8 :=, int9 :=, int10 :=, Bypass := #FALSE, commands := "Unit1.Em4.HmiInterface".cmAnodeMainPnP2AxisX.commands, interlockOk := "Unit1.Em4.ControlNodes".cm.Interlock.anodeMainPnP2AxisX.source.posAbsolute, intOut := "Unit1.Em4.HmiInterface".intCondition.Axis_06.Position.intOut)
   END_RUNG
   RUNG wire#powerrail
      Contact( "Unit1.Em4.ControlNodes".emRelations.em7.cmStatus.sepaClampBottomUpDown.inWorkPos )
   END_RUNG wire#w1
   RUNG wire#powerrail
      Contact( #TRUE )
   END_RUNG wire#w1
   RUNG wire#powerrail
      I_Contact( "Unit1.Em4.ControlNodes".emRelations.em7.softCam.sepaGripperAxisX.anodePnPZonePos.inPos )
   END_RUNG wire#w2
   RUNG wire#powerrail
      Contact( #TRUE )
   END_RUNG wire#w2
   RUNG wire#powerrail
      I_Contact( "Unit1.Em4.ControlNodes".mainPnP."step".action1[1070] )
      I_Contact( "Unit1.Em4.ControlNodes".mainPnP."step".action1[130] )
      I_Contact( "Unit1.Em4.ControlNodes".mainPnP."step".action1[150] )
      I_Contact( "Unit1.Em4.ControlNodes".mainPnP."step".action1[220] )
      I_Contact( "Unit1.Em4.ControlNodes".mainPnP."step".action1[720] )
      Not()
      wire#w3
      Contact( "Unit1.Em4.ControlNodes".cm.Interlock.anodeMainPnP2AxisX.source.posAbsolute[0] )
      Move(in := 0, out1 => "Unit1.Em4.ControlNodes".cmAnodeMainPnP2AxisX.commands.selectSetPosition)
      Coil( "Unit1.Em4.ControlNodes".cm.axisCommand.anodeMainPnP2AxisX.posAbsolute[0] )
   END_RUNG
   RUNG wire#powerrail
      I_Contact( "Unit1.Em4.ControlNodes".gaugeRnR."step".action1[110] )
      I_Contact( "Unit1.Em4.ControlNodes".gaugeRnR."step".action1[520] )
      I_Contact( "Unit1.Em4.ControlNodes".gaugeRnR."step".action1[1120] )
      I_Contact( "Unit1.Em4.ControlNodes".gaugeRnR."step".action1[1520] )
      I_Contact( "Unit1.Em4.ControlNodes".gaugeRnR."step".action1[2120] )
      I_Contact( "Unit1.Em4.ControlNodes".gaugeRnR."step".action1[2520] )
      I_Contact( "Unit1.Em4.ControlNodes".gaugeRnR."step".action1[3210] )
      Not()
   END_RUNG wire#w3
   // the same network as SCL:
   #"AnodeMainPnP2AxisX Position_"[0](Status := #unitStatus,   // "Position.LER_Axis"
                           int1 := "Unit1.Em4.ControlNodes".cm.softCam.anodeMainPnP2AxisZ.upPos.inPos,
                           int2 := "Unit1.Em4.ControlNodes".cm.softCam.anodeMainPnP1AxisX.reelCutConveyerPos.inPos,
                           int3 := "Unit1.Em4.ControlNodes".emRelations.em7.cmStatus.sepaClampBottomUpDown.inWorkPos OR #TRUE,
                           int4 := "Unit1.Em4.ControlNodes".cmAnodeNgPnp1stFwdBwd.monitoring.inHomePos,
                           int5 := "Unit1.Em4.ControlNodes".cmAnodeNgPnp2ndFwdBwd.monitoring.inHomePos,
                           int6 := NOT "Unit1.Em4.ControlNodes".emRelations.em7.softCam.sepaGripperAxisX.anodePnPZonePos.inPos OR #TRUE,
                           Bypass := #FALSE,
                           commands := "Unit1.Em4.HmiInterface".cmAnodeMainPnP2AxisX.commands,
                           interlockOk := "Unit1.Em4.ControlNodes".cm.Interlock.anodeMainPnP2AxisX.source.posAbsolute,
                           intOut := "Unit1.Em4.HmiInterface".intCondition.Axis_06.Position.intOut);
   #_w1 := (NOT (NOT "Unit1.Em4.ControlNodes".mainPnP."step".action1[1070] AND NOT "Unit1.Em4.ControlNodes".mainPnP."step".action1[130] AND NOT "Unit1.Em4.ControlNodes".mainPnP."step".action1[150] AND NOT "Unit1.Em4.ControlNodes".mainPnP."step".action1[220] AND NOT "Unit1.Em4.ControlNodes".mainPnP."step".action1[720]) OR NOT (NOT "Unit1.Em4.ControlNodes".gaugeRnR."step".action1[110] AND NOT "Unit1.Em4.ControlNodes".gaugeRnR."step".action1[520] AND NOT "Unit1.Em4.ControlNodes".gaugeRnR."step".action1[1120] AND NOT "Unit1.Em4.ControlNodes".gaugeRnR."step".action1[1520] AND NOT "Unit1.Em4.ControlNodes".gaugeRnR."step".action1[2120] AND NOT "Unit1.Em4.ControlNodes".gaugeRnR."step".action1[2520] AND NOT "Unit1.Em4.ControlNodes".gaugeRnR."step".action1[3210])) AND "Unit1.Em4.ControlNodes".cm.Interlock.anodeMainPnP2AxisX.source.posAbsolute[0];
   IF #_w1 THEN "Unit1.Em4.ControlNodes".cmAnodeMainPnP2AxisX.commands.selectSetPosition := 0; END_IF;
   "Unit1.Em4.ControlNodes".cm.axisCommand.anodeMainPnP2AxisX.posAbsolute[0] := #_w1;
END_REGION

REGION Network 137: CmAnodeMainPnP2AxisX Position Absolute Position1
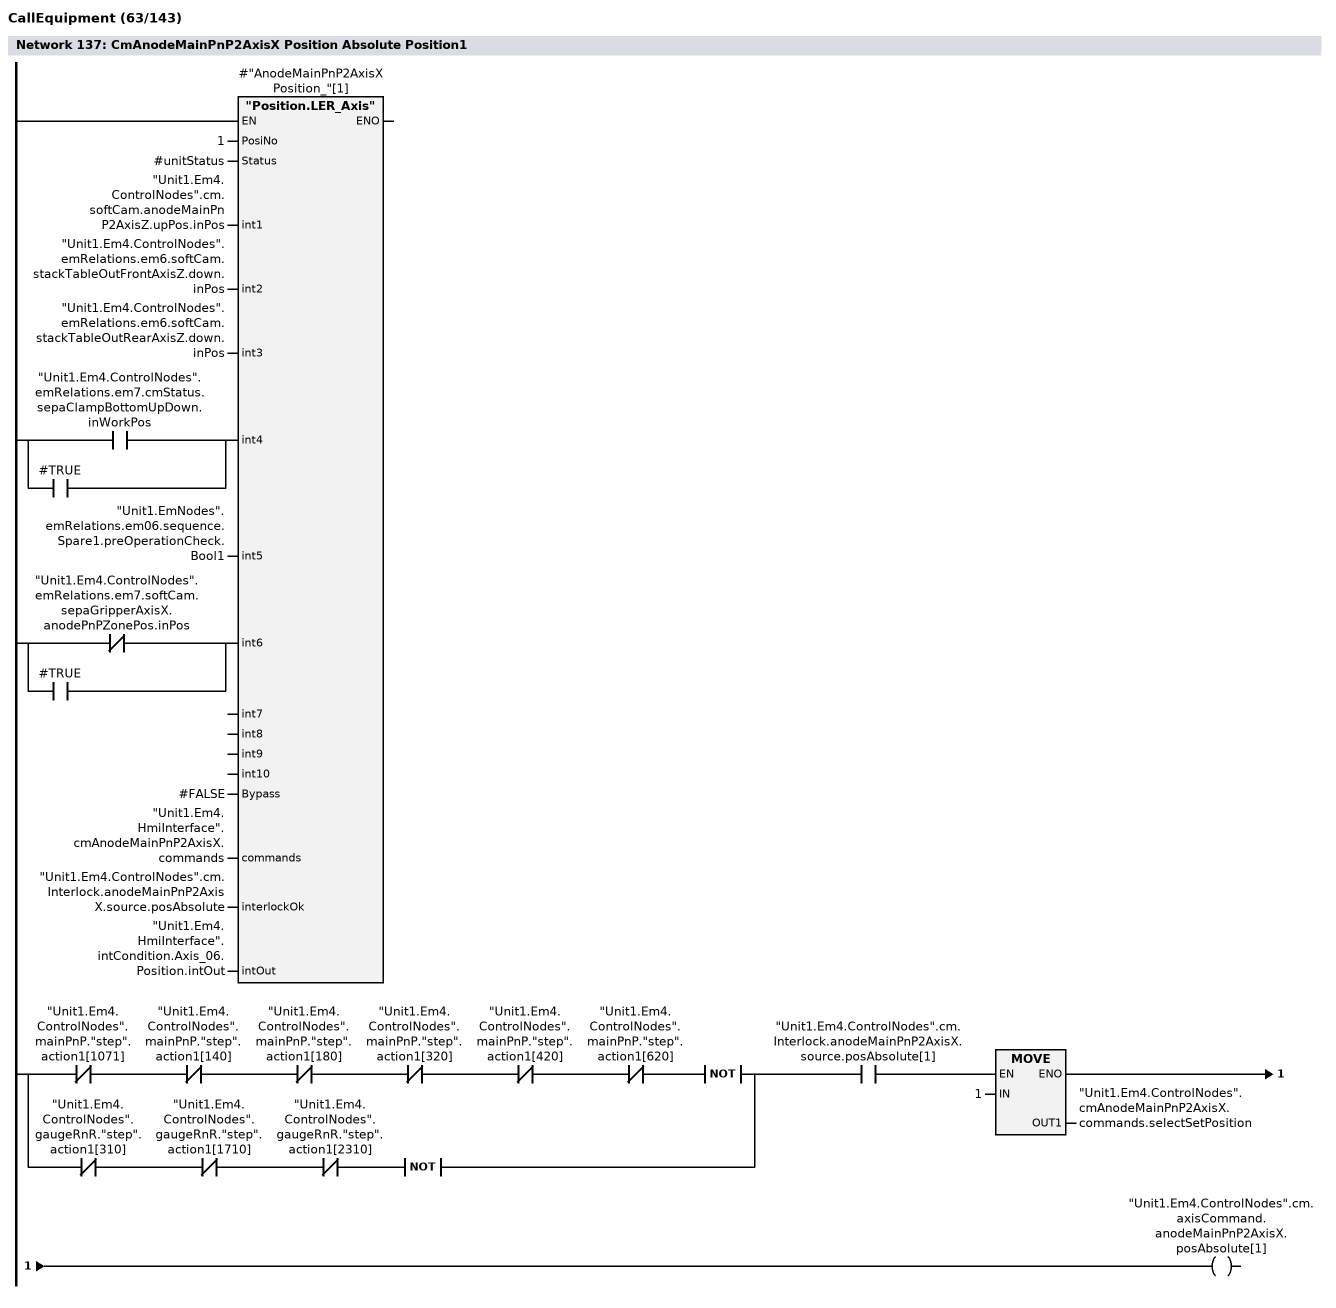
   RUNG wire#powerrail
      #"AnodeMainPnP2AxisX Position_"[1](int4 := wire#w1, int6 := wire#w2, PosiNo := 1, Status := #unitStatus, int1 := "Unit1.Em4.ControlNodes".cm.softCam.anodeMainPnP2AxisZ.upPos.inPos, int2 := "Unit1.Em4.ControlNodes".emRelations.em6.softCam.stackTableOutFrontAxisZ.down.inPos, int3 := "Unit1.Em4.ControlNodes".emRelations.em6.softCam.stackTableOutRearAxisZ.down.inPos, int5 := "Unit1.EmNodes".emRelations.em06.sequence.Spare1.preOperationCheck.Bool1, int7 :=, int8 :=, int9 :=, int10 :=, Bypass := #FALSE, commands := "Unit1.Em4.HmiInterface".cmAnodeMainPnP2AxisX.commands, interlockOk := "Unit1.Em4.ControlNodes".cm.Interlock.anodeMainPnP2AxisX.source.posAbsolute, intOut := "Unit1.Em4.HmiInterface".intCondition.Axis_06.Position.intOut)
   END_RUNG
   RUNG wire#powerrail
      Contact( "Unit1.Em4.ControlNodes".emRelations.em7.cmStatus.sepaClampBottomUpDown.inWorkPos )
   END_RUNG wire#w1
   RUNG wire#powerrail
      Contact( #TRUE )
   END_RUNG wire#w1
   RUNG wire#powerrail
      I_Contact( "Unit1.Em4.ControlNodes".emRelations.em7.softCam.sepaGripperAxisX.anodePnPZonePos.inPos )
   END_RUNG wire#w2
   RUNG wire#powerrail
      Contact( #TRUE )
   END_RUNG wire#w2
   RUNG wire#powerrail
      I_Contact( "Unit1.Em4.ControlNodes".mainPnP."step".action1[1071] )
      I_Contact( "Unit1.Em4.ControlNodes".mainPnP."step".action1[140] )
      I_Contact( "Unit1.Em4.ControlNodes".mainPnP."step".action1[180] )
      I_Contact( "Unit1.Em4.ControlNodes".mainPnP."step".action1[320] )
      I_Contact( "Unit1.Em4.ControlNodes".mainPnP."step".action1[420] )
      I_Contact( "Unit1.Em4.ControlNodes".mainPnP."step".action1[620] )
      Not()
      wire#w3
      Contact( "Unit1.Em4.ControlNodes".cm.Interlock.anodeMainPnP2AxisX.source.posAbsolute[1] )
      Move(in := 1, out1 => "Unit1.Em4.ControlNodes".cmAnodeMainPnP2AxisX.commands.selectSetPosition)
      Coil( "Unit1.Em4.ControlNodes".cm.axisCommand.anodeMainPnP2AxisX.posAbsolute[1] )
   END_RUNG
   RUNG wire#powerrail
      I_Contact( "Unit1.Em4.ControlNodes".gaugeRnR."step".action1[310] )
      I_Contact( "Unit1.Em4.ControlNodes".gaugeRnR."step".action1[1710] )
      I_Contact( "Unit1.Em4.ControlNodes".gaugeRnR."step".action1[2310] )
      Not()
   END_RUNG wire#w3
   // the same network as SCL:
   #"AnodeMainPnP2AxisX Position_"[1](PosiNo := 1,   // "Position.LER_Axis"
                           Status := #unitStatus,
                           int1 := "Unit1.Em4.ControlNodes".cm.softCam.anodeMainPnP2AxisZ.upPos.inPos,
                           int2 := "Unit1.Em4.ControlNodes".emRelations.em6.softCam.stackTableOutFrontAxisZ.down.inPos,
                           int3 := "Unit1.Em4.ControlNodes".emRelations.em6.softCam.stackTableOutRearAxisZ.down.inPos,
                           int4 := "Unit1.Em4.ControlNodes".emRelations.em7.cmStatus.sepaClampBottomUpDown.inWorkPos OR #TRUE,
                           int5 := "Unit1.EmNodes".emRelations.em06.sequence.Spare1.preOperationCheck.Bool1,
                           int6 := NOT "Unit1.Em4.ControlNodes".emRelations.em7.softCam.sepaGripperAxisX.anodePnPZonePos.inPos OR #TRUE,
                           Bypass := #FALSE,
                           commands := "Unit1.Em4.HmiInterface".cmAnodeMainPnP2AxisX.commands,
                           interlockOk := "Unit1.Em4.ControlNodes".cm.Interlock.anodeMainPnP2AxisX.source.posAbsolute,
                           intOut := "Unit1.Em4.HmiInterface".intCondition.Axis_06.Position.intOut);
   #_w1 := (NOT (NOT "Unit1.Em4.ControlNodes".mainPnP."step".action1[1071] AND NOT "Unit1.Em4.ControlNodes".mainPnP."step".action1[140] AND NOT "Unit1.Em4.ControlNodes".mainPnP."step".action1[180] AND NOT "Unit1.Em4.ControlNodes".mainPnP."step".action1[320] AND NOT "Unit1.Em4.ControlNodes".mainPnP."step".action1[420] AND NOT "Unit1.Em4.ControlNodes".mainPnP."step".action1[620]) OR NOT (NOT "Unit1.Em4.ControlNodes".gaugeRnR."step".action1[310] AND NOT "Unit1.Em4.ControlNodes".gaugeRnR."step".action1[1710] AND NOT "Unit1.Em4.ControlNodes".gaugeRnR."step".action1[2310])) AND "Unit1.Em4.ControlNodes".cm.Interlock.anodeMainPnP2AxisX.source.posAbsolute[1];
   IF #_w1 THEN "Unit1.Em4.ControlNodes".cmAnodeMainPnP2AxisX.commands.selectSetPosition := 1; END_IF;
   "Unit1.Em4.ControlNodes".cm.axisCommand.anodeMainPnP2AxisX.posAbsolute[1] := #_w1;
END_REGION

REGION Network 138: CmAnodeMainPnP2AxisX Position Absolute Position2
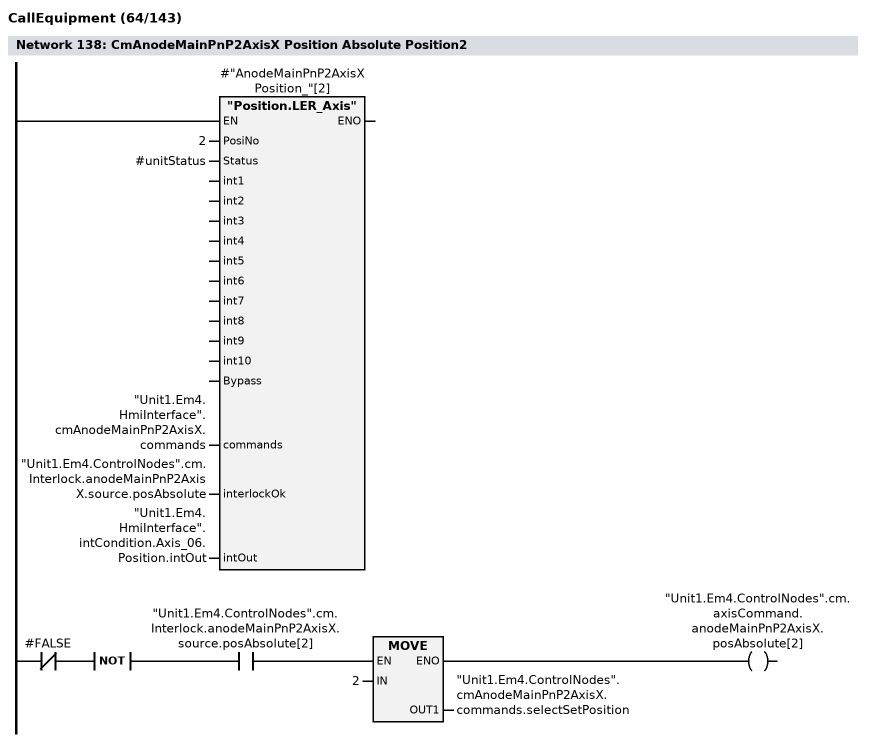
   RUNG wire#powerrail
      #"AnodeMainPnP2AxisX Position_"[2](PosiNo := 2, Status := #unitStatus, int1 :=, int2 :=, int3 :=, int4 :=, int5 :=, int6 :=, int7 :=, int8 :=, int9 :=, int10 :=, Bypass :=, commands := "Unit1.Em4.HmiInterface".cmAnodeMainPnP2AxisX.commands, interlockOk := "Unit1.Em4.ControlNodes".cm.Interlock.anodeMainPnP2AxisX.source.posAbsolute, intOut := "Unit1.Em4.HmiInterface".intCondition.Axis_06.Position.intOut)
   END_RUNG
   RUNG wire#powerrail
      I_Contact( #FALSE )
      Not()
      Contact( "Unit1.Em4.ControlNodes".cm.Interlock.anodeMainPnP2AxisX.source.posAbsolute[2] )
      Move(in := 2, out1 => "Unit1.Em4.ControlNodes".cmAnodeMainPnP2AxisX.commands.selectSetPosition)
      Coil( "Unit1.Em4.ControlNodes".cm.axisCommand.anodeMainPnP2AxisX.posAbsolute[2] )
   END_RUNG
   // the same network as SCL:
   #"AnodeMainPnP2AxisX Position_"[2](PosiNo := 2,   // "Position.LER_Axis"
                           Status := #unitStatus,
                           commands := "Unit1.Em4.HmiInterface".cmAnodeMainPnP2AxisX.commands,
                           interlockOk := "Unit1.Em4.ControlNodes".cm.Interlock.anodeMainPnP2AxisX.source.posAbsolute,
                           intOut := "Unit1.Em4.HmiInterface".intCondition.Axis_06.Position.intOut);
   #_w1 := NOT (NOT #FALSE) AND "Unit1.Em4.ControlNodes".cm.Interlock.anodeMainPnP2AxisX.source.posAbsolute[2];
   IF #_w1 THEN "Unit1.Em4.ControlNodes".cmAnodeMainPnP2AxisX.commands.selectSetPosition := 2; END_IF;
   "Unit1.Em4.ControlNodes".cm.axisCommand.anodeMainPnP2AxisX.posAbsolute[2] := #_w1;
END_REGION

REGION Network 139: CmAnodeMainPnP2AxisX Position Absolute Position3
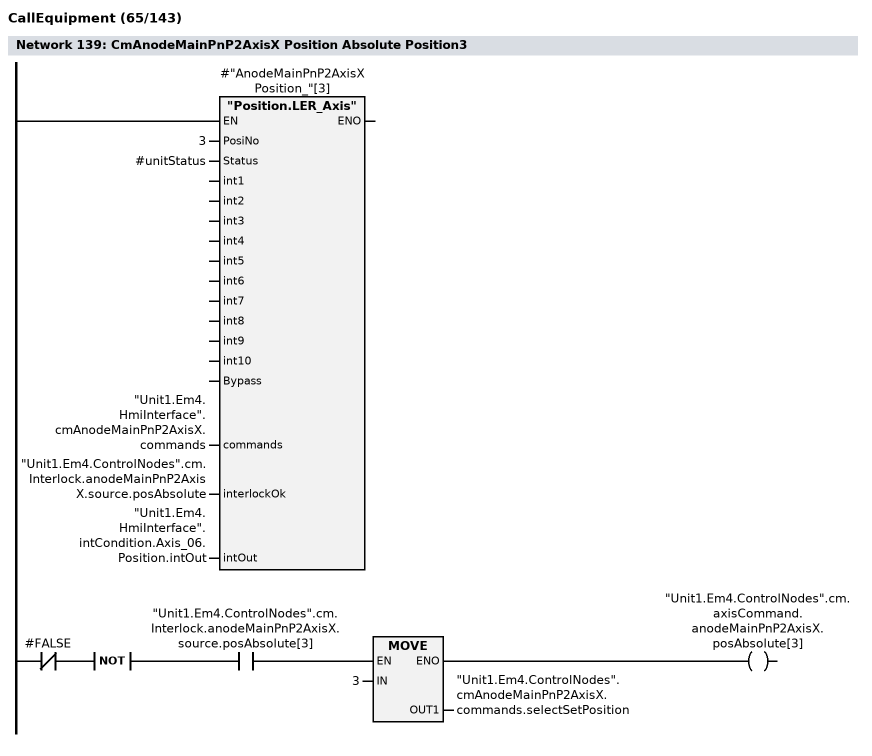
   RUNG wire#powerrail
      #"AnodeMainPnP2AxisX Position_"[3](PosiNo := 3, Status := #unitStatus, int1 :=, int2 :=, int3 :=, int4 :=, int5 :=, int6 :=, int7 :=, int8 :=, int9 :=, int10 :=, Bypass :=, commands := "Unit1.Em4.HmiInterface".cmAnodeMainPnP2AxisX.commands, interlockOk := "Unit1.Em4.ControlNodes".cm.Interlock.anodeMainPnP2AxisX.source.posAbsolute, intOut := "Unit1.Em4.HmiInterface".intCondition.Axis_06.Position.intOut)
   END_RUNG
   RUNG wire#powerrail
      I_Contact( #FALSE )
      Not()
      Contact( "Unit1.Em4.ControlNodes".cm.Interlock.anodeMainPnP2AxisX.source.posAbsolute[3] )
      Move(in := 3, out1 => "Unit1.Em4.ControlNodes".cmAnodeMainPnP2AxisX.commands.selectSetPosition)
      Coil( "Unit1.Em4.ControlNodes".cm.axisCommand.anodeMainPnP2AxisX.posAbsolute[3] )
   END_RUNG
   // the same network as SCL:
   #"AnodeMainPnP2AxisX Position_"[3](PosiNo := 3,   // "Position.LER_Axis"
                           Status := #unitStatus,
                           commands := "Unit1.Em4.HmiInterface".cmAnodeMainPnP2AxisX.commands,
                           interlockOk := "Unit1.Em4.ControlNodes".cm.Interlock.anodeMainPnP2AxisX.source.posAbsolute,
                           intOut := "Unit1.Em4.HmiInterface".intCondition.Axis_06.Position.intOut);
   #_w1 := NOT (NOT #FALSE) AND "Unit1.Em4.ControlNodes".cm.Interlock.anodeMainPnP2AxisX.source.posAbsolute[3];
   IF #_w1 THEN "Unit1.Em4.ControlNodes".cmAnodeMainPnP2AxisX.commands.selectSetPosition := 3; END_IF;
   "Unit1.Em4.ControlNodes".cm.axisCommand.anodeMainPnP2AxisX.posAbsolute[3] := #_w1;
END_REGION

REGION Network 140: CmAnodeMainPnP2AxisX Position Absolute Position4
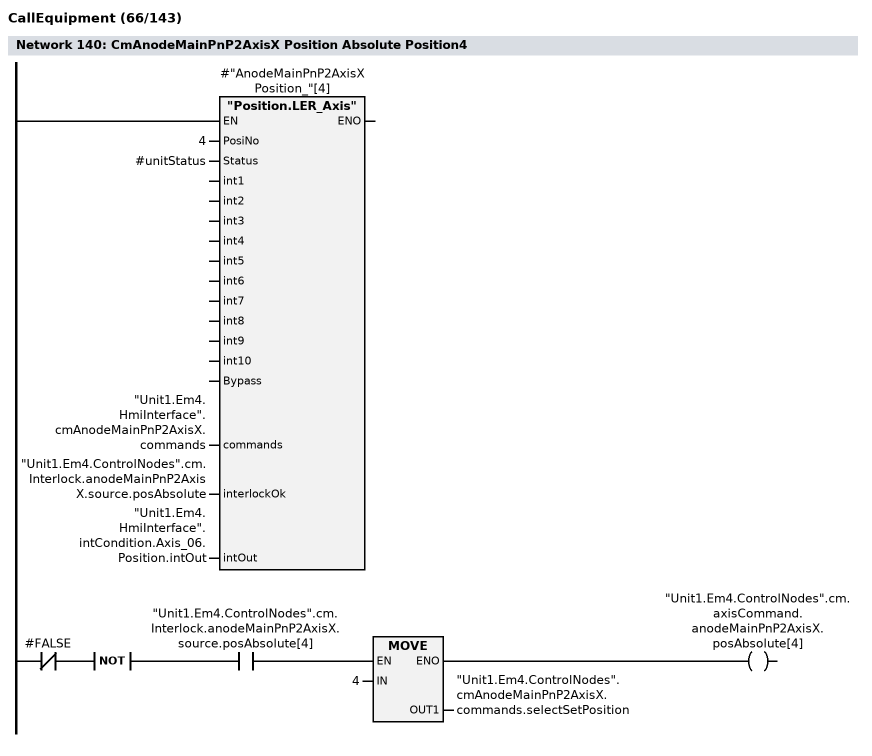
   RUNG wire#powerrail
      #"AnodeMainPnP2AxisX Position_"[4](PosiNo := 4, Status := #unitStatus, int1 :=, int2 :=, int3 :=, int4 :=, int5 :=, int6 :=, int7 :=, int8 :=, int9 :=, int10 :=, Bypass :=, commands := "Unit1.Em4.HmiInterface".cmAnodeMainPnP2AxisX.commands, interlockOk := "Unit1.Em4.ControlNodes".cm.Interlock.anodeMainPnP2AxisX.source.posAbsolute, intOut := "Unit1.Em4.HmiInterface".intCondition.Axis_06.Position.intOut)
   END_RUNG
   RUNG wire#powerrail
      I_Contact( #FALSE )
      Not()
      Contact( "Unit1.Em4.ControlNodes".cm.Interlock.anodeMainPnP2AxisX.source.posAbsolute[4] )
      Move(in := 4, out1 => "Unit1.Em4.ControlNodes".cmAnodeMainPnP2AxisX.commands.selectSetPosition)
      Coil( "Unit1.Em4.ControlNodes".cm.axisCommand.anodeMainPnP2AxisX.posAbsolute[4] )
   END_RUNG
   // the same network as SCL:
   #"AnodeMainPnP2AxisX Position_"[4](PosiNo := 4,   // "Position.LER_Axis"
                           Status := #unitStatus,
                           commands := "Unit1.Em4.HmiInterface".cmAnodeMainPnP2AxisX.commands,
                           interlockOk := "Unit1.Em4.ControlNodes".cm.Interlock.anodeMainPnP2AxisX.source.posAbsolute,
                           intOut := "Unit1.Em4.HmiInterface".intCondition.Axis_06.Position.intOut);
   #_w1 := NOT (NOT #FALSE) AND "Unit1.Em4.ControlNodes".cm.Interlock.anodeMainPnP2AxisX.source.posAbsolute[4];
   IF #_w1 THEN "Unit1.Em4.ControlNodes".cmAnodeMainPnP2AxisX.commands.selectSetPosition := 4; END_IF;
   "Unit1.Em4.ControlNodes".cm.axisCommand.anodeMainPnP2AxisX.posAbsolute[4] := #_w1;
END_REGION

REGION Network 141: CmAnodeMainPnP2AxisX Position Absolute Position5
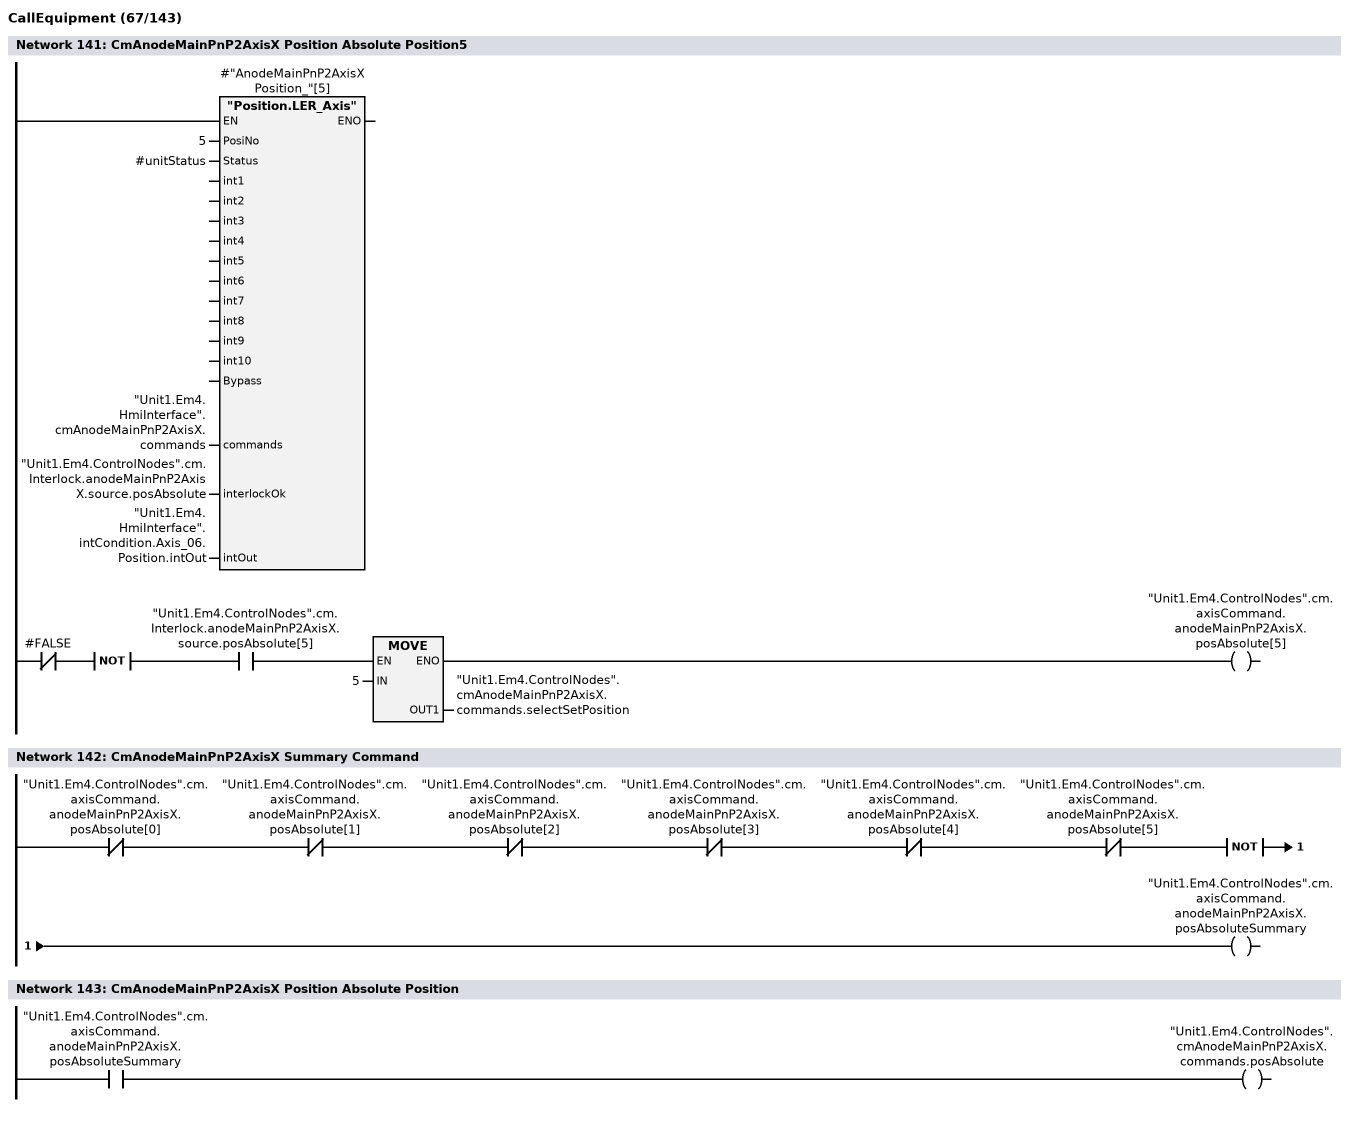
   RUNG wire#powerrail
      #"AnodeMainPnP2AxisX Position_"[5](PosiNo := 5, Status := #unitStatus, int1 :=, int2 :=, int3 :=, int4 :=, int5 :=, int6 :=, int7 :=, int8 :=, int9 :=, int10 :=, Bypass :=, commands := "Unit1.Em4.HmiInterface".cmAnodeMainPnP2AxisX.commands, interlockOk := "Unit1.Em4.ControlNodes".cm.Interlock.anodeMainPnP2AxisX.source.posAbsolute, intOut := "Unit1.Em4.HmiInterface".intCondition.Axis_06.Position.intOut)
   END_RUNG
   RUNG wire#powerrail
      I_Contact( #FALSE )
      Not()
      Contact( "Unit1.Em4.ControlNodes".cm.Interlock.anodeMainPnP2AxisX.source.posAbsolute[5] )
      Move(in := 5, out1 => "Unit1.Em4.ControlNodes".cmAnodeMainPnP2AxisX.commands.selectSetPosition)
      Coil( "Unit1.Em4.ControlNodes".cm.axisCommand.anodeMainPnP2AxisX.posAbsolute[5] )
   END_RUNG
   // the same network as SCL:
   #"AnodeMainPnP2AxisX Position_"[5](PosiNo := 5,   // "Position.LER_Axis"
                           Status := #unitStatus,
                           commands := "Unit1.Em4.HmiInterface".cmAnodeMainPnP2AxisX.commands,
                           interlockOk := "Unit1.Em4.ControlNodes".cm.Interlock.anodeMainPnP2AxisX.source.posAbsolute,
                           intOut := "Unit1.Em4.HmiInterface".intCondition.Axis_06.Position.intOut);
   #_w1 := NOT (NOT #FALSE) AND "Unit1.Em4.ControlNodes".cm.Interlock.anodeMainPnP2AxisX.source.posAbsolute[5];
   IF #_w1 THEN "Unit1.Em4.ControlNodes".cmAnodeMainPnP2AxisX.commands.selectSetPosition := 5; END_IF;
   "Unit1.Em4.ControlNodes".cm.axisCommand.anodeMainPnP2AxisX.posAbsolute[5] := #_w1;
END_REGION

REGION Network 142: CmAnodeMainPnP2AxisX Summary Command
   RUNG wire#powerrail
      I_Contact( "Unit1.Em4.ControlNodes".cm.axisCommand.anodeMainPnP2AxisX.posAbsolute[0] )
      I_Contact( "Unit1.Em4.ControlNodes".cm.axisCommand.anodeMainPnP2AxisX.posAbsolute[1] )
      I_Contact( "Unit1.Em4.ControlNodes".cm.axisCommand.anodeMainPnP2AxisX.posAbsolute[2] )
      I_Contact( "Unit1.Em4.ControlNodes".cm.axisCommand.anodeMainPnP2AxisX.posAbsolute[3] )
      I_Contact( "Unit1.Em4.ControlNodes".cm.axisCommand.anodeMainPnP2AxisX.posAbsolute[4] )
      I_Contact( "Unit1.Em4.ControlNodes".cm.axisCommand.anodeMainPnP2AxisX.posAbsolute[5] )
      Not()
      Coil( "Unit1.Em4.ControlNodes".cm.axisCommand.anodeMainPnP2AxisX.posAbsoluteSummary )
   END_RUNG
   // the same network as SCL:
   "Unit1.Em4.ControlNodes".cm.axisCommand.anodeMainPnP2AxisX.posAbsoluteSummary := NOT (NOT "Unit1.Em4.ControlNodes".cm.axisCommand.anodeMainPnP2AxisX.posAbsolute[0] AND NOT "Unit1.Em4.ControlNodes".cm.axisCommand.anodeMainPnP2AxisX.posAbsolute[1] AND NOT "Unit1.Em4.ControlNodes".cm.axisCommand.anodeMainPnP2AxisX.posAbsolute[2] AND NOT "Unit1.Em4.ControlNodes".cm.axisCommand.anodeMainPnP2AxisX.posAbsolute[3] AND NOT "Unit1.Em4.ControlNodes".cm.axisCommand.anodeMainPnP2AxisX.posAbsolute[4] AND NOT "Unit1.Em4.ControlNodes".cm.axisCommand.anodeMainPnP2AxisX.posAbsolute[5]);
END_REGION

REGION Network 143: CmAnodeMainPnP2AxisX Position Absolute Position
   RUNG wire#powerrail
      Contact( "Unit1.Em4.ControlNodes".cm.axisCommand.anodeMainPnP2AxisX.posAbsoluteSummary )
      Coil( "Unit1.Em4.ControlNodes".cmAnodeMainPnP2AxisX.commands.posAbsolute )
   END_RUNG
   // the same network as SCL:
   "Unit1.Em4.ControlNodes".cmAnodeMainPnP2AxisX.commands.posAbsolute := "Unit1.Em4.ControlNodes".cm.axisCommand.anodeMainPnP2AxisX.posAbsoluteSummary;
END_REGION

REGION Network 144: CmAnodeMainPnP2AxisX Interlock Summary
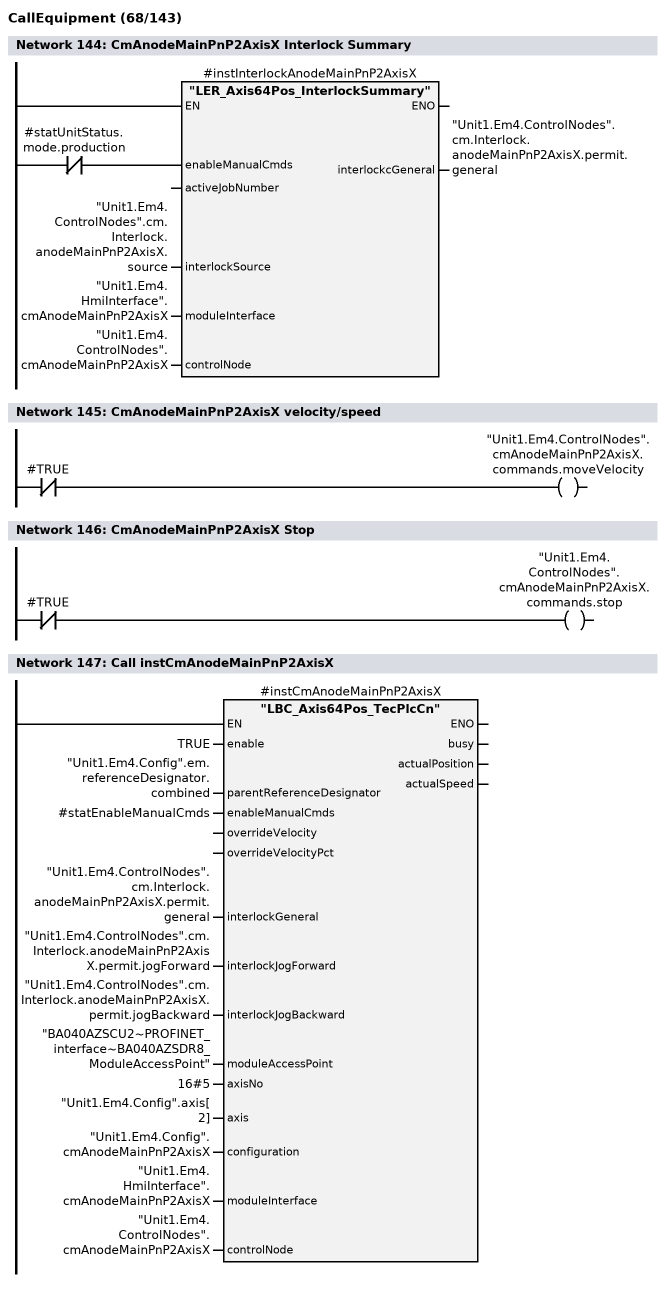
   RUNG wire#powerrail
      #instInterlockAnodeMainPnP2AxisX(enableManualCmds := wire#w1, activeJobNumber :=, interlockSource := "Unit1.Em4.ControlNodes".cm.Interlock.anodeMainPnP2AxisX.source, moduleInterface := "Unit1.Em4.HmiInterface".cmAnodeMainPnP2AxisX, controlNode := "Unit1.Em4.ControlNodes".cmAnodeMainPnP2AxisX, interlockcGeneral => "Unit1.Em4.ControlNodes".cm.Interlock.anodeMainPnP2AxisX.permit.general)
   END_RUNG
   RUNG wire#powerrail
      I_Contact( #statUnitStatus.mode.production )
   END_RUNG wire#w1
   // the same network as SCL:
   #instInterlockAnodeMainPnP2AxisX(enableManualCmds := NOT #statUnitStatus.mode.production,   // "LER_Axis64Pos_InterlockSummary"
                           interlockSource := "Unit1.Em4.ControlNodes".cm.Interlock.anodeMainPnP2AxisX.source,
                           moduleInterface := "Unit1.Em4.HmiInterface".cmAnodeMainPnP2AxisX,
                           controlNode := "Unit1.Em4.ControlNodes".cmAnodeMainPnP2AxisX,
                           interlockcGeneral => "Unit1.Em4.ControlNodes".cm.Interlock.anodeMainPnP2AxisX.permit.general);
END_REGION

REGION Network 145: CmAnodeMainPnP2AxisX velocity/speed
   RUNG wire#powerrail
      I_Contact( #TRUE )
      Coil( "Unit1.Em4.ControlNodes".cmAnodeMainPnP2AxisX.commands.moveVelocity )
   END_RUNG
   // the same network as SCL:
   "Unit1.Em4.ControlNodes".cmAnodeMainPnP2AxisX.commands.moveVelocity := NOT #TRUE;
END_REGION

REGION Network 146: CmAnodeMainPnP2AxisX Stop
   RUNG wire#powerrail
      I_Contact( #TRUE )
      Coil( "Unit1.Em4.ControlNodes".cmAnodeMainPnP2AxisX.commands.stop )
   END_RUNG
   // the same network as SCL:
   "Unit1.Em4.ControlNodes".cmAnodeMainPnP2AxisX.commands.stop := NOT #TRUE;
END_REGION

REGION Network 147: Call instCmAnodeMainPnP2AxisX
   RUNG wire#powerrail
      #instCmAnodeMainPnP2AxisX(enable := TRUE, parentReferenceDesignator := "Unit1.Em4.Config".em.referenceDesignator.combined, enableManualCmds := #statEnableManualCmds, overrideVelocity :=, overrideVelocityPct :=, interlockGeneral := "Unit1.Em4.ControlNodes".cm.Interlock.anodeMainPnP2AxisX.permit.general, interlockJogForward := "Unit1.Em4.ControlNodes".cm.Interlock.anodeMainPnP2AxisX.permit.jogForward, interlockJogBackward := "Unit1.Em4.ControlNodes".cm.Interlock.anodeMainPnP2AxisX.permit.jogBackward, moduleAccessPoint := "BA040AZSCU2~PROFINET_interface~BA040AZSDR8_ModuleAccessPoint", axisNo := 16#5, axis := "Unit1.Em4.Config".axis[2], configuration := "Unit1.Em4.Config".cmAnodeMainPnP2AxisX, moduleInterface := "Unit1.Em4.HmiInterface".cmAnodeMainPnP2AxisX, controlNode := "Unit1.Em4.ControlNodes".cmAnodeMainPnP2AxisX, busy =>, actualPosition =>, actualSpeed =>)
   END_RUNG
   // the same network as SCL:
   #instCmAnodeMainPnP2AxisX(enable := TRUE,   // "LBC_Axis64Pos_TecPlcCn"
                           parentReferenceDesignator := "Unit1.Em4.Config".em.referenceDesignator.combined,
                           enableManualCmds := #statEnableManualCmds,
                           interlockGeneral := "Unit1.Em4.ControlNodes".cm.Interlock.anodeMainPnP2AxisX.permit.general,
                           interlockJogForward := "Unit1.Em4.ControlNodes".cm.Interlock.anodeMainPnP2AxisX.permit.jogForward,
                           interlockJogBackward := "Unit1.Em4.ControlNodes".cm.Interlock.anodeMainPnP2AxisX.permit.jogBackward,
                           moduleAccessPoint := "BA040AZSCU2~PROFINET_interface~BA040AZSDR8_ModuleAccessPoint",
                           axisNo := 16#5,
                           axis := "Unit1.Em4.Config".axis[2],
                           configuration := "Unit1.Em4.Config".cmAnodeMainPnP2AxisX,
                           moduleInterface := "Unit1.Em4.HmiInterface".cmAnodeMainPnP2AxisX,
                           controlNode := "Unit1.Em4.ControlNodes".cmAnodeMainPnP2AxisX);
END_REGION

REGION Network 148: CmAnodeMainPnP2AxisX SoftCam
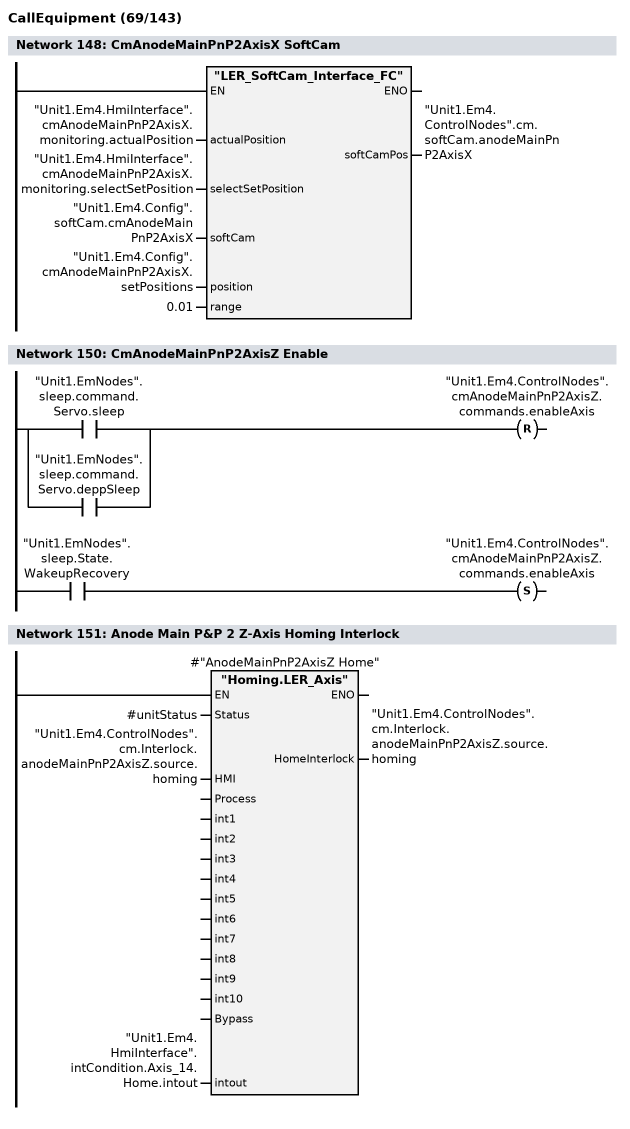
   RUNG wire#powerrail
      "LER_SoftCam_Interface_FC"(actualPosition := "Unit1.Em4.HmiInterface".cmAnodeMainPnP2AxisX.monitoring.actualPosition, selectSetPosition := "Unit1.Em4.HmiInterface".cmAnodeMainPnP2AxisX.monitoring.selectSetPosition, softCam := "Unit1.Em4.Config".softCam.cmAnodeMainPnP2AxisX, position := "Unit1.Em4.Config".cmAnodeMainPnP2AxisX.setPositions, range := 0.01, softCamPos => "Unit1.Em4.ControlNodes".cm.softCam.anodeMainPnP2AxisX)
   END_RUNG
   // the same network as SCL:
   "LER_SoftCam_Interface_FC"(actualPosition := "Unit1.Em4.HmiInterface".cmAnodeMainPnP2AxisX.monitoring.actualPosition,
                           selectSetPosition := "Unit1.Em4.HmiInterface".cmAnodeMainPnP2AxisX.monitoring.selectSetPosition,
                           softCam := "Unit1.Em4.Config".softCam.cmAnodeMainPnP2AxisX,
                           position := "Unit1.Em4.Config".cmAnodeMainPnP2AxisX.setPositions,
                           range := 0.01,
                           softCamPos => "Unit1.Em4.ControlNodes".cm.softCam.anodeMainPnP2AxisX);
END_REGION

REGION Network 150: CmAnodeMainPnP2AxisZ Enable
   RUNG wire#powerrail
      Contact( "Unit1.EmNodes".sleep.command.Servo.sleep )
      wire#w1
      R_Coil( "Unit1.Em4.ControlNodes".cmAnodeMainPnP2AxisZ.commands.enableAxis )
   END_RUNG
   RUNG wire#powerrail
      Contact( "Unit1.EmNodes".sleep.command.Servo.deppSleep )
   END_RUNG wire#w1
   RUNG wire#powerrail
      Contact( "Unit1.EmNodes".sleep.State.WakeupRecovery )
      S_Coil( "Unit1.Em4.ControlNodes".cmAnodeMainPnP2AxisZ.commands.enableAxis )
   END_RUNG
   // the same network as SCL:
   IF "Unit1.EmNodes".sleep.command.Servo.sleep OR "Unit1.EmNodes".sleep.command.Servo.deppSleep THEN
       "Unit1.Em4.ControlNodes".cmAnodeMainPnP2AxisZ.commands.enableAxis := FALSE;
   END_IF;
   IF "Unit1.EmNodes".sleep.State.WakeupRecovery THEN
       "Unit1.Em4.ControlNodes".cmAnodeMainPnP2AxisZ.commands.enableAxis := TRUE;
   END_IF;
END_REGION

REGION Network 151: Anode Main P&P 2 Z-Axis Homing Interlock
   RUNG wire#powerrail
      #"AnodeMainPnP2AxisZ Home"(Status := #unitStatus, HMI := "Unit1.Em4.ControlNodes".cm.Interlock.anodeMainPnP2AxisZ.source.homing, Process :=, int1 :=, int2 :=, int3 :=, int4 :=, int5 :=, int6 :=, int7 :=, int8 :=, int9 :=, int10 :=, Bypass :=, intout := "Unit1.Em4.HmiInterface".intCondition.Axis_14.Home.intout, HomeInterlock => "Unit1.Em4.ControlNodes".cm.Interlock.anodeMainPnP2AxisZ.source.homing)
   END_RUNG
   // the same network as SCL:
   #"AnodeMainPnP2AxisZ Home"(Status := #unitStatus,   // "Homing.LER_Axis"
                           HMI := "Unit1.Em4.ControlNodes".cm.Interlock.anodeMainPnP2AxisZ.source.homing,
                           intout := "Unit1.Em4.HmiInterface".intCondition.Axis_14.Home.intout,
                           HomeInterlock => "Unit1.Em4.ControlNodes".cm.Interlock.anodeMainPnP2AxisZ.source.homing);
END_REGION

REGION Network 152: CmAnodeMainPnP2AxisZ Position Absolute Jog
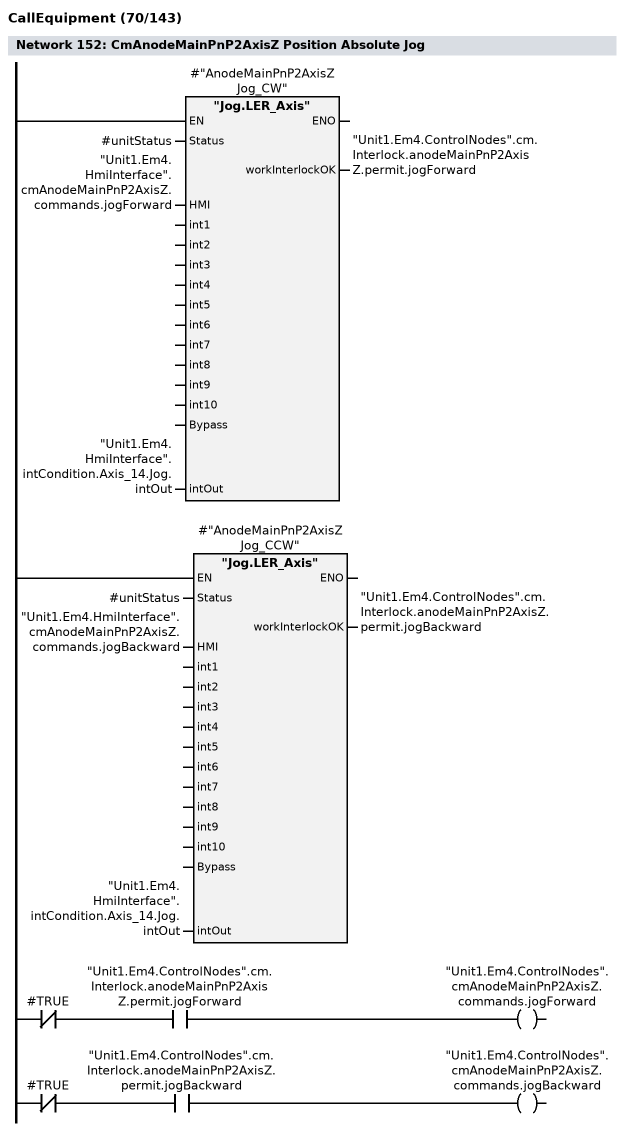
   RUNG wire#powerrail
      #"AnodeMainPnP2AxisZ Jog_CW"(Status := #unitStatus, HMI := "Unit1.Em4.HmiInterface".cmAnodeMainPnP2AxisZ.commands.jogForward, int1 :=, int2 :=, int3 :=, int4 :=, int5 :=, int6 :=, int7 :=, int8 :=, int9 :=, int10 :=, Bypass :=, intOut := "Unit1.Em4.HmiInterface".intCondition.Axis_14.Jog.intOut, workInterlockOK => "Unit1.Em4.ControlNodes".cm.Interlock.anodeMainPnP2AxisZ.permit.jogForward)
   END_RUNG
   RUNG wire#powerrail
      #"AnodeMainPnP2AxisZ Jog_CCW"(Status := #unitStatus, HMI := "Unit1.Em4.HmiInterface".cmAnodeMainPnP2AxisZ.commands.jogBackward, int1 :=, int2 :=, int3 :=, int4 :=, int5 :=, int6 :=, int7 :=, int8 :=, int9 :=, int10 :=, Bypass :=, intOut := "Unit1.Em4.HmiInterface".intCondition.Axis_14.Jog.intOut, workInterlockOK => "Unit1.Em4.ControlNodes".cm.Interlock.anodeMainPnP2AxisZ.permit.jogBackward)
   END_RUNG
   RUNG wire#powerrail
      I_Contact( #TRUE )
      Contact( "Unit1.Em4.ControlNodes".cm.Interlock.anodeMainPnP2AxisZ.permit.jogForward )
      Coil( "Unit1.Em4.ControlNodes".cmAnodeMainPnP2AxisZ.commands.jogForward )
   END_RUNG
   RUNG wire#powerrail
      I_Contact( #TRUE )
      Contact( "Unit1.Em4.ControlNodes".cm.Interlock.anodeMainPnP2AxisZ.permit.jogBackward )
      Coil( "Unit1.Em4.ControlNodes".cmAnodeMainPnP2AxisZ.commands.jogBackward )
   END_RUNG
   // the same network as SCL:
   #"AnodeMainPnP2AxisZ Jog_CW"(Status := #unitStatus,   // "Jog.LER_Axis"
                           HMI := "Unit1.Em4.HmiInterface".cmAnodeMainPnP2AxisZ.commands.jogForward,
                           intOut := "Unit1.Em4.HmiInterface".intCondition.Axis_14.Jog.intOut,
                           workInterlockOK => "Unit1.Em4.ControlNodes".cm.Interlock.anodeMainPnP2AxisZ.permit.jogForward);
   #"AnodeMainPnP2AxisZ Jog_CCW"(Status := #unitStatus,   // "Jog.LER_Axis"
                           HMI := "Unit1.Em4.HmiInterface".cmAnodeMainPnP2AxisZ.commands.jogBackward,
                           intOut := "Unit1.Em4.HmiInterface".intCondition.Axis_14.Jog.intOut,
                           workInterlockOK => "Unit1.Em4.ControlNodes".cm.Interlock.anodeMainPnP2AxisZ.permit.jogBackward);
   "Unit1.Em4.ControlNodes".cmAnodeMainPnP2AxisZ.commands.jogForward := NOT #TRUE AND "Unit1.Em4.ControlNodes".cm.Interlock.anodeMainPnP2AxisZ.permit.jogForward;
   "Unit1.Em4.ControlNodes".cmAnodeMainPnP2AxisZ.commands.jogBackward := NOT #TRUE AND "Unit1.Em4.ControlNodes".cm.Interlock.anodeMainPnP2AxisZ.permit.jogBackward;
END_REGION

REGION Network 153: CmAnodeMainPnP2AxisZ Position Absolute Position0
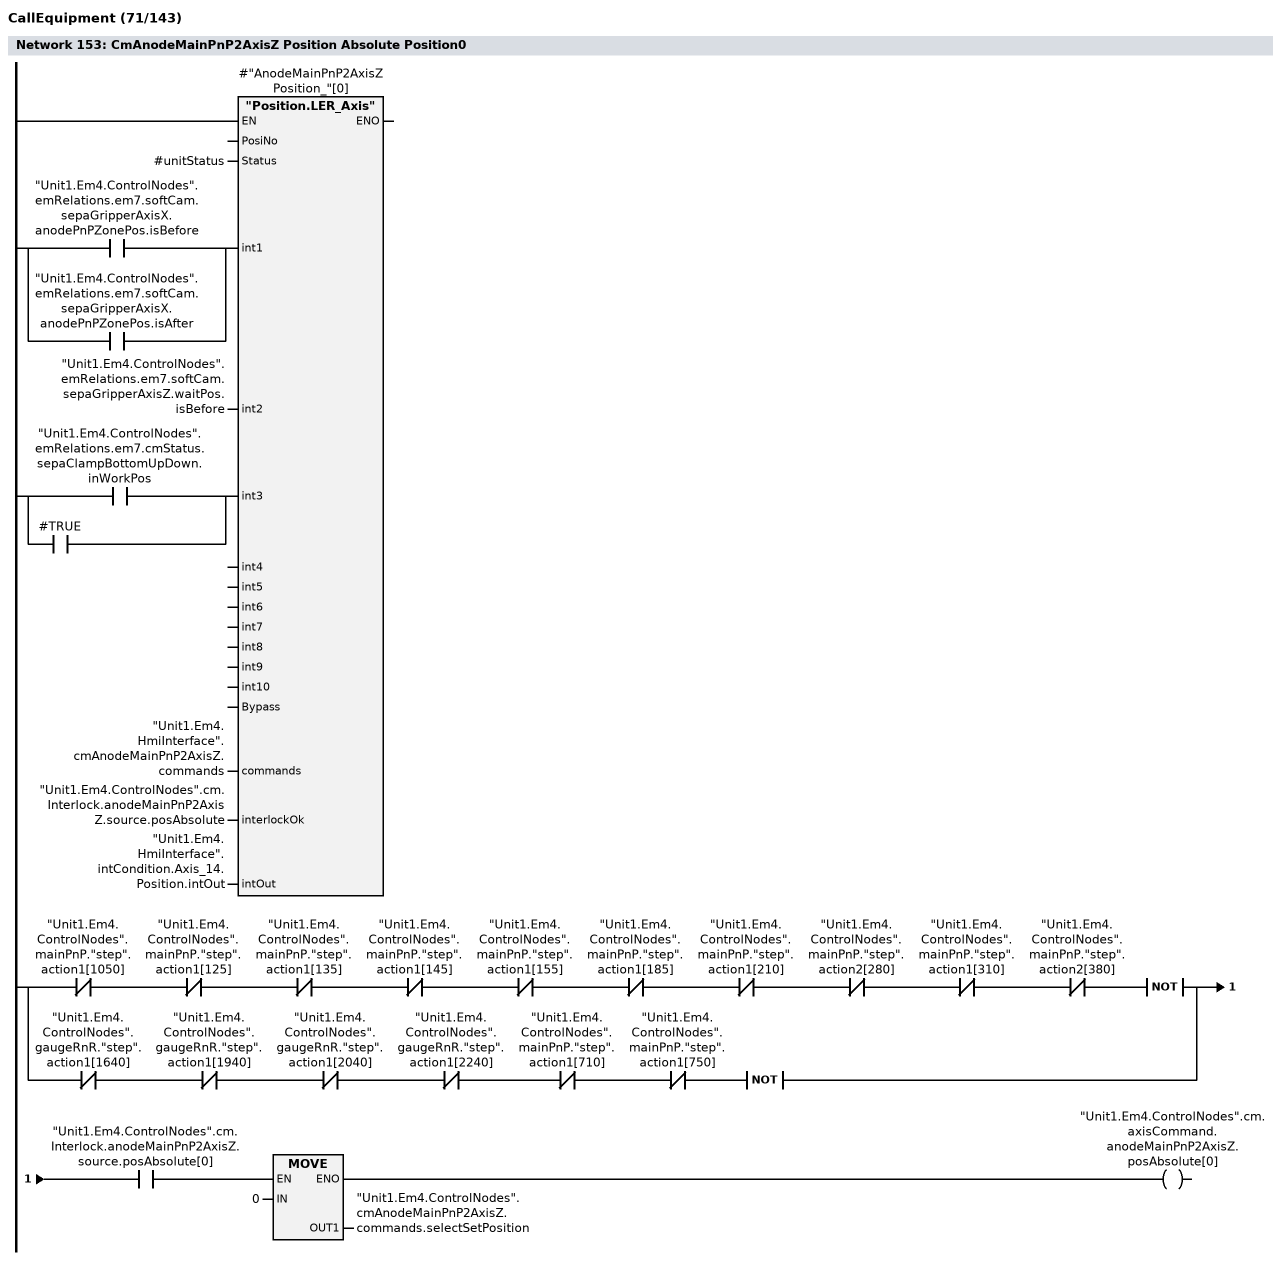
   RUNG wire#powerrail
      #"AnodeMainPnP2AxisZ Position_"[0](int1 := wire#w1, int3 := wire#w2, PosiNo :=, Status := #unitStatus, int2 := "Unit1.Em4.ControlNodes".emRelations.em7.softCam.sepaGripperAxisZ.waitPos.isBefore, int4 :=, int5 :=, int6 :=, int7 :=, int8 :=, int9 :=, int10 :=, Bypass :=, commands := "Unit1.Em4.HmiInterface".cmAnodeMainPnP2AxisZ.commands, interlockOk := "Unit1.Em4.ControlNodes".cm.Interlock.anodeMainPnP2AxisZ.source.posAbsolute, intOut := "Unit1.Em4.HmiInterface".intCondition.Axis_14.Position.intOut)
   END_RUNG
   RUNG wire#powerrail
      Contact( "Unit1.Em4.ControlNodes".emRelations.em7.softCam.sepaGripperAxisX.anodePnPZonePos.isBefore )
   END_RUNG wire#w1
   RUNG wire#powerrail
      Contact( "Unit1.Em4.ControlNodes".emRelations.em7.softCam.sepaGripperAxisX.anodePnPZonePos.isAfter )
   END_RUNG wire#w1
   RUNG wire#powerrail
      Contact( "Unit1.Em4.ControlNodes".emRelations.em7.cmStatus.sepaClampBottomUpDown.inWorkPos )
   END_RUNG wire#w2
   RUNG wire#powerrail
      Contact( #TRUE )
   END_RUNG wire#w2
   RUNG wire#powerrail
      I_Contact( "Unit1.Em4.ControlNodes".mainPnP."step".action1[1050] )
      I_Contact( "Unit1.Em4.ControlNodes".mainPnP."step".action1[125] )
      I_Contact( "Unit1.Em4.ControlNodes".mainPnP."step".action1[135] )
      I_Contact( "Unit1.Em4.ControlNodes".mainPnP."step".action1[145] )
      I_Contact( "Unit1.Em4.ControlNodes".mainPnP."step".action1[155] )
      I_Contact( "Unit1.Em4.ControlNodes".mainPnP."step".action1[185] )
      I_Contact( "Unit1.Em4.ControlNodes".mainPnP."step".action1[210] )
      I_Contact( "Unit1.Em4.ControlNodes".mainPnP."step".action2[280] )
      I_Contact( "Unit1.Em4.ControlNodes".mainPnP."step".action1[310] )
      I_Contact( "Unit1.Em4.ControlNodes".mainPnP."step".action2[380] )
      Not()
      wire#w3
      Contact( "Unit1.Em4.ControlNodes".cm.Interlock.anodeMainPnP2AxisZ.source.posAbsolute[0] )
      Move(in := 0, out1 => "Unit1.Em4.ControlNodes".cmAnodeMainPnP2AxisZ.commands.selectSetPosition)
      Coil( "Unit1.Em4.ControlNodes".cm.axisCommand.anodeMainPnP2AxisZ.posAbsolute[0] )
   END_RUNG
   RUNG wire#powerrail
      I_Contact( "Unit1.Em4.ControlNodes".gaugeRnR."step".action1[1640] )
      I_Contact( "Unit1.Em4.ControlNodes".gaugeRnR."step".action1[1940] )
      I_Contact( "Unit1.Em4.ControlNodes".gaugeRnR."step".action1[2040] )
      I_Contact( "Unit1.Em4.ControlNodes".gaugeRnR."step".action1[2240] )
      I_Contact( "Unit1.Em4.ControlNodes".mainPnP."step".action1[710] )
      I_Contact( "Unit1.Em4.ControlNodes".mainPnP."step".action1[750] )
      Not()
   END_RUNG wire#w3
   // the same network as SCL:
   #"AnodeMainPnP2AxisZ Position_"[0](Status := #unitStatus,   // "Position.LER_Axis"
                           int1 := "Unit1.Em4.ControlNodes".emRelations.em7.softCam.sepaGripperAxisX.anodePnPZonePos.isBefore OR "Unit1.Em4.ControlNodes".emRelations.em7.softCam.sepaGripperAxisX.anodePnPZonePos.isAfter,
                           int2 := "Unit1.Em4.ControlNodes".emRelations.em7.softCam.sepaGripperAxisZ.waitPos.isBefore,
                           int3 := "Unit1.Em4.ControlNodes".emRelations.em7.cmStatus.sepaClampBottomUpDown.inWorkPos OR #TRUE,
                           commands := "Unit1.Em4.HmiInterface".cmAnodeMainPnP2AxisZ.commands,
                           interlockOk := "Unit1.Em4.ControlNodes".cm.Interlock.anodeMainPnP2AxisZ.source.posAbsolute,
                           intOut := "Unit1.Em4.HmiInterface".intCondition.Axis_14.Position.intOut);
   #_w1 := (NOT (NOT "Unit1.Em4.ControlNodes".mainPnP."step".action1[1050] AND NOT "Unit1.Em4.ControlNodes".mainPnP."step".action1[125] AND NOT "Unit1.Em4.ControlNodes".mainPnP."step".action1[135] AND NOT "Unit1.Em4.ControlNodes".mainPnP."step".action1[145] AND NOT "Unit1.Em4.ControlNodes".mainPnP."step".action1[155] AND NOT "Unit1.Em4.ControlNodes".mainPnP."step".action1[185] AND NOT "Unit1.Em4.ControlNodes".mainPnP."step".action1[210] AND NOT "Unit1.Em4.ControlNodes".mainPnP."step".action2[280] AND NOT "Unit1.Em4.ControlNodes".mainPnP."step".action1[310] AND NOT "Unit1.Em4.ControlNodes".mainPnP."step".action2[380]) OR NOT (NOT "Unit1.Em4.ControlNodes".gaugeRnR."step".action1[1640] AND NOT "Unit1.Em4.ControlNodes".gaugeRnR."step".action1[1940] AND NOT "Unit1.Em4.ControlNodes".gaugeRnR."step".action1[2040] AND NOT "Unit1.Em4.ControlNodes".gaugeRnR."step".action1[2240] AND NOT "Unit1.Em4.ControlNodes".mainPnP."step".action1[710] AND NOT "Unit1.Em4.ControlNodes".mainPnP."step".action1[750])) AND "Unit1.Em4.ControlNodes".cm.Interlock.anodeMainPnP2AxisZ.source.posAbsolute[0];
   IF #_w1 THEN "Unit1.Em4.ControlNodes".cmAnodeMainPnP2AxisZ.commands.selectSetPosition := 0; END_IF;
   "Unit1.Em4.ControlNodes".cm.axisCommand.anodeMainPnP2AxisZ.posAbsolute[0] := #_w1;
END_REGION

REGION Network 154: CmAnodeMainPnP2AxisZ Position Absolute Position1
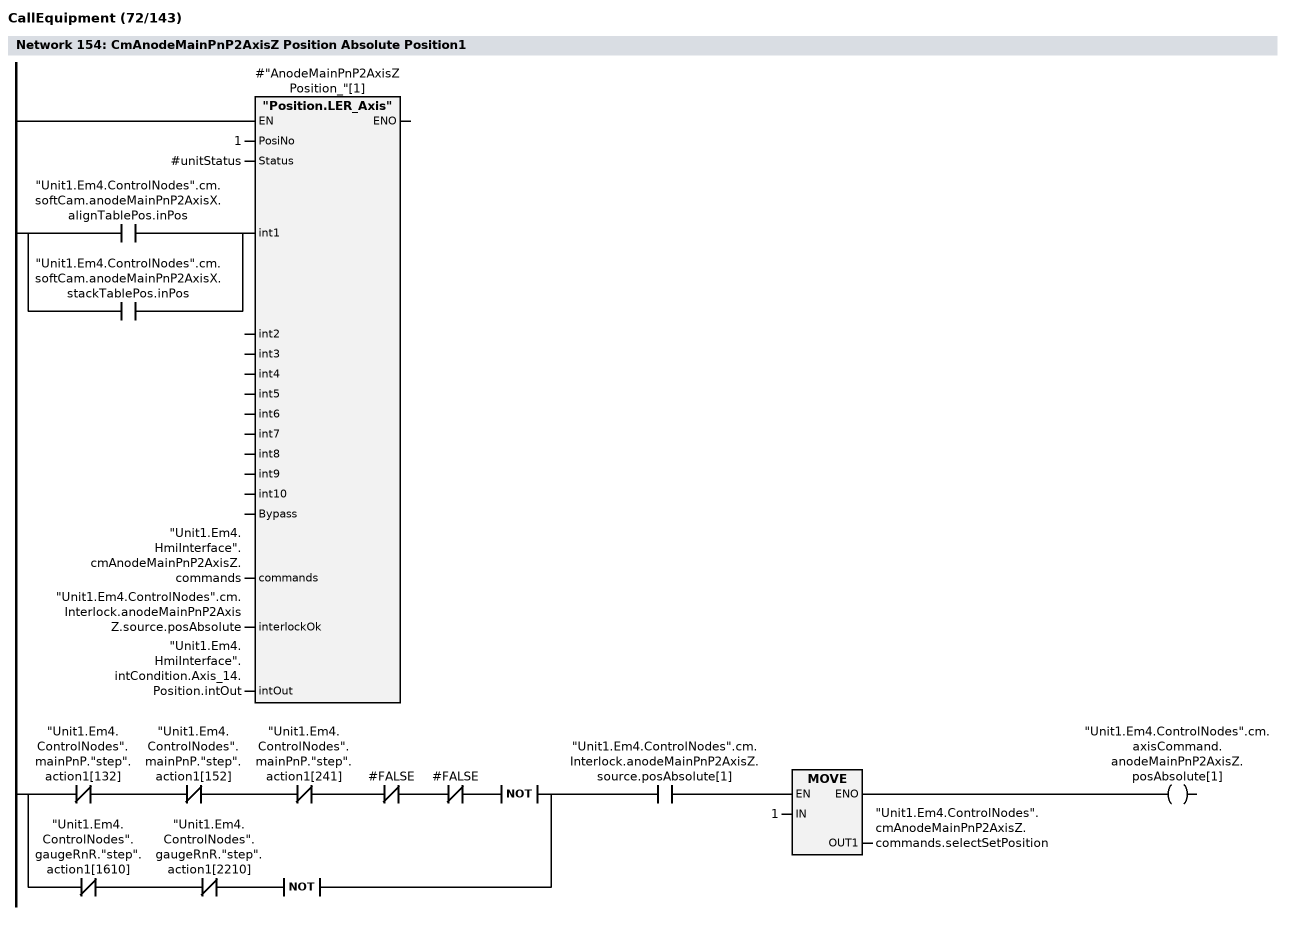
   RUNG wire#powerrail
      #"AnodeMainPnP2AxisZ Position_"[1](int1 := wire#w1, PosiNo := 1, Status := #unitStatus, int2 :=, int3 :=, int4 :=, int5 :=, int6 :=, int7 :=, int8 :=, int9 :=, int10 :=, Bypass :=, commands := "Unit1.Em4.HmiInterface".cmAnodeMainPnP2AxisZ.commands, interlockOk := "Unit1.Em4.ControlNodes".cm.Interlock.anodeMainPnP2AxisZ.source.posAbsolute, intOut := "Unit1.Em4.HmiInterface".intCondition.Axis_14.Position.intOut)
   END_RUNG
   RUNG wire#powerrail
      Contact( "Unit1.Em4.ControlNodes".cm.softCam.anodeMainPnP2AxisX.alignTablePos.inPos )
   END_RUNG wire#w1
   RUNG wire#powerrail
      Contact( "Unit1.Em4.ControlNodes".cm.softCam.anodeMainPnP2AxisX.stackTablePos.inPos )
   END_RUNG wire#w1
   RUNG wire#powerrail
      I_Contact( "Unit1.Em4.ControlNodes".mainPnP."step".action1[132] )
      I_Contact( "Unit1.Em4.ControlNodes".mainPnP."step".action1[152] )
      I_Contact( "Unit1.Em4.ControlNodes".mainPnP."step".action1[241] )
      I_Contact( #FALSE )
      I_Contact( #FALSE )
      Not()
      wire#w2
      Contact( "Unit1.Em4.ControlNodes".cm.Interlock.anodeMainPnP2AxisZ.source.posAbsolute[1] )
      Move(in := 1, out1 => "Unit1.Em4.ControlNodes".cmAnodeMainPnP2AxisZ.commands.selectSetPosition)
      Coil( "Unit1.Em4.ControlNodes".cm.axisCommand.anodeMainPnP2AxisZ.posAbsolute[1] )
   END_RUNG
   RUNG wire#powerrail
      I_Contact( "Unit1.Em4.ControlNodes".gaugeRnR."step".action1[1610] )
      I_Contact( "Unit1.Em4.ControlNodes".gaugeRnR."step".action1[2210] )
      Not()
   END_RUNG wire#w2
   // the same network as SCL:
   #"AnodeMainPnP2AxisZ Position_"[1](PosiNo := 1,   // "Position.LER_Axis"
                           Status := #unitStatus,
                           int1 := "Unit1.Em4.ControlNodes".cm.softCam.anodeMainPnP2AxisX.alignTablePos.inPos OR "Unit1.Em4.ControlNodes".cm.softCam.anodeMainPnP2AxisX.stackTablePos.inPos,
                           commands := "Unit1.Em4.HmiInterface".cmAnodeMainPnP2AxisZ.commands,
                           interlockOk := "Unit1.Em4.ControlNodes".cm.Interlock.anodeMainPnP2AxisZ.source.posAbsolute,
                           intOut := "Unit1.Em4.HmiInterface".intCondition.Axis_14.Position.intOut);
   #_w1 := (NOT (NOT "Unit1.Em4.ControlNodes".mainPnP."step".action1[132] AND NOT "Unit1.Em4.ControlNodes".mainPnP."step".action1[152] AND NOT "Unit1.Em4.ControlNodes".mainPnP."step".action1[241] AND NOT #FALSE AND NOT #FALSE) OR NOT (NOT "Unit1.Em4.ControlNodes".gaugeRnR."step".action1[1610] AND NOT "Unit1.Em4.ControlNodes".gaugeRnR."step".action1[2210])) AND "Unit1.Em4.ControlNodes".cm.Interlock.anodeMainPnP2AxisZ.source.posAbsolute[1];
   IF #_w1 THEN "Unit1.Em4.ControlNodes".cmAnodeMainPnP2AxisZ.commands.selectSetPosition := 1; END_IF;
   "Unit1.Em4.ControlNodes".cm.axisCommand.anodeMainPnP2AxisZ.posAbsolute[1] := #_w1;
END_REGION

REGION Network 155: CmAnodeMainPnP2AxisZ Position Absolute Position2
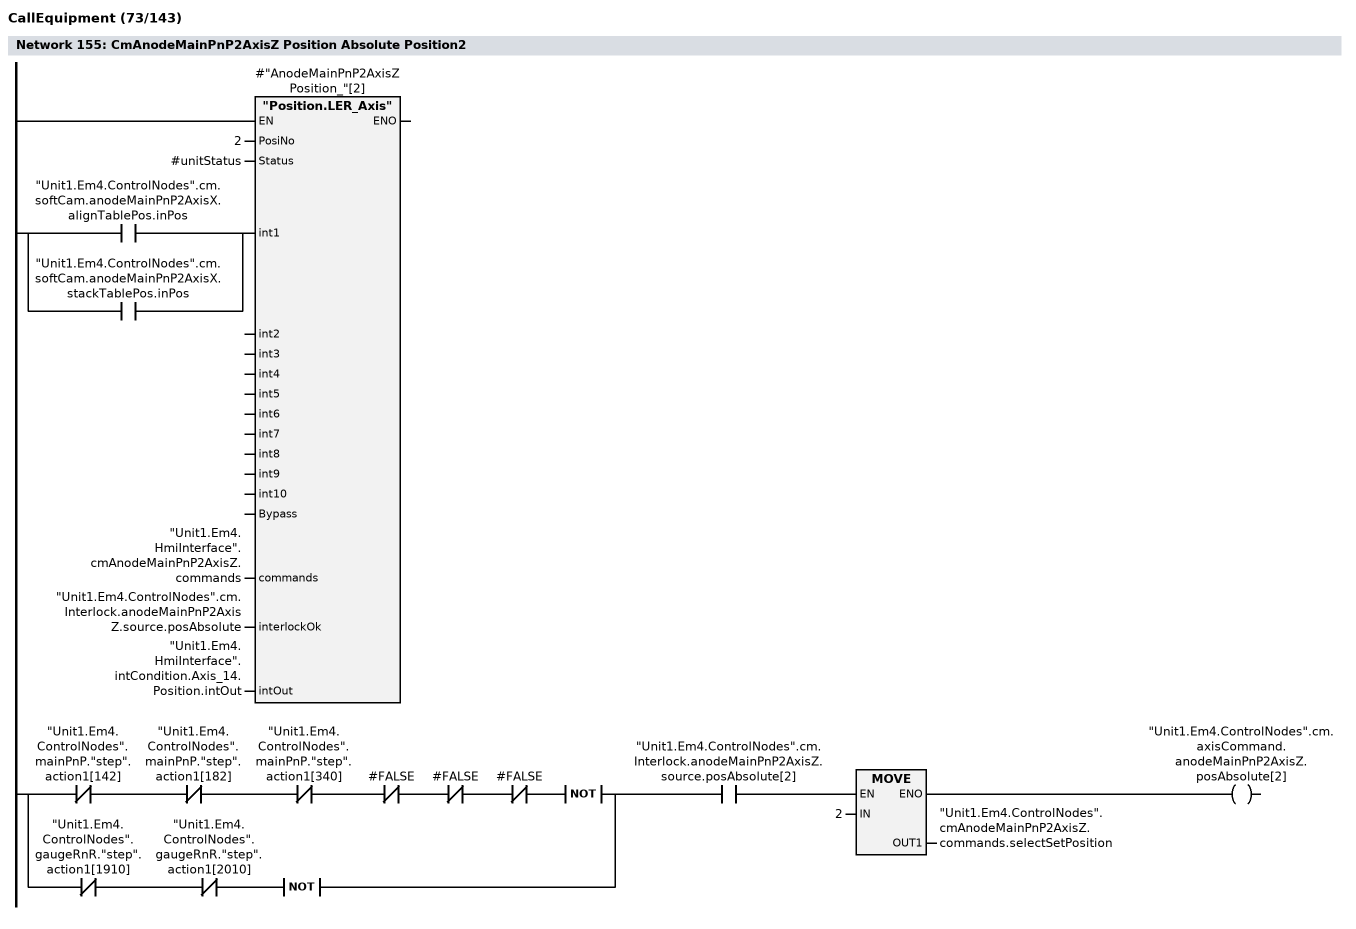
   RUNG wire#powerrail
      #"AnodeMainPnP2AxisZ Position_"[2](int1 := wire#w1, PosiNo := 2, Status := #unitStatus, int2 :=, int3 :=, int4 :=, int5 :=, int6 :=, int7 :=, int8 :=, int9 :=, int10 :=, Bypass :=, commands := "Unit1.Em4.HmiInterface".cmAnodeMainPnP2AxisZ.commands, interlockOk := "Unit1.Em4.ControlNodes".cm.Interlock.anodeMainPnP2AxisZ.source.posAbsolute, intOut := "Unit1.Em4.HmiInterface".intCondition.Axis_14.Position.intOut)
   END_RUNG
   RUNG wire#powerrail
      Contact( "Unit1.Em4.ControlNodes".cm.softCam.anodeMainPnP2AxisX.alignTablePos.inPos )
   END_RUNG wire#w1
   RUNG wire#powerrail
      Contact( "Unit1.Em4.ControlNodes".cm.softCam.anodeMainPnP2AxisX.stackTablePos.inPos )
   END_RUNG wire#w1
   RUNG wire#powerrail
      I_Contact( "Unit1.Em4.ControlNodes".mainPnP."step".action1[142] )
      I_Contact( "Unit1.Em4.ControlNodes".mainPnP."step".action1[182] )
      I_Contact( "Unit1.Em4.ControlNodes".mainPnP."step".action1[340] )
      I_Contact( #FALSE )
      I_Contact( #FALSE )
      I_Contact( #FALSE )
      Not()
      wire#w2
      Contact( "Unit1.Em4.ControlNodes".cm.Interlock.anodeMainPnP2AxisZ.source.posAbsolute[2] )
      Move(in := 2, out1 => "Unit1.Em4.ControlNodes".cmAnodeMainPnP2AxisZ.commands.selectSetPosition)
      Coil( "Unit1.Em4.ControlNodes".cm.axisCommand.anodeMainPnP2AxisZ.posAbsolute[2] )
   END_RUNG
   RUNG wire#powerrail
      I_Contact( "Unit1.Em4.ControlNodes".gaugeRnR."step".action1[1910] )
      I_Contact( "Unit1.Em4.ControlNodes".gaugeRnR."step".action1[2010] )
      Not()
   END_RUNG wire#w2
   // the same network as SCL:
   #"AnodeMainPnP2AxisZ Position_"[2](PosiNo := 2,   // "Position.LER_Axis"
                           Status := #unitStatus,
                           int1 := "Unit1.Em4.ControlNodes".cm.softCam.anodeMainPnP2AxisX.alignTablePos.inPos OR "Unit1.Em4.ControlNodes".cm.softCam.anodeMainPnP2AxisX.stackTablePos.inPos,
                           commands := "Unit1.Em4.HmiInterface".cmAnodeMainPnP2AxisZ.commands,
                           interlockOk := "Unit1.Em4.ControlNodes".cm.Interlock.anodeMainPnP2AxisZ.source.posAbsolute,
                           intOut := "Unit1.Em4.HmiInterface".intCondition.Axis_14.Position.intOut);
   #_w1 := (NOT (NOT "Unit1.Em4.ControlNodes".mainPnP."step".action1[142] AND NOT "Unit1.Em4.ControlNodes".mainPnP."step".action1[182] AND NOT "Unit1.Em4.ControlNodes".mainPnP."step".action1[340] AND NOT #FALSE AND NOT #FALSE AND NOT #FALSE) OR NOT (NOT "Unit1.Em4.ControlNodes".gaugeRnR."step".action1[1910] AND NOT "Unit1.Em4.ControlNodes".gaugeRnR."step".action1[2010])) AND "Unit1.Em4.ControlNodes".cm.Interlock.anodeMainPnP2AxisZ.source.posAbsolute[2];
   IF #_w1 THEN "Unit1.Em4.ControlNodes".cmAnodeMainPnP2AxisZ.commands.selectSetPosition := 2; END_IF;
   "Unit1.Em4.ControlNodes".cm.axisCommand.anodeMainPnP2AxisZ.posAbsolute[2] := #_w1;
END_REGION

REGION Network 156: CmAnodeMainPnP2AxisZ Position Absolute Position3
